// TwinCAT 3 PLC project Kid_PLC_Universal
// ProgramVersion: 3.1.4022.0
// libraries:
//   Tc2_EtherCAT, * (Beckhoff Automation GmbH)
//   Tc2_Math, * (Beckhoff Automation GmbH)
//   Tc2_MC2, * (Beckhoff Automation GmbH)
//   Tc2_System, * (Beckhoff Automation GmbH)
//   Tc2_SystemCX, * (Beckhoff Automation GmbH)
//   Tc2_Utilities, * (Beckhoff Automation GmbH)
//   Tc3_Interfaces, * (Beckhoff Automation GmbH)
//   Tc3_Module, * (Beckhoff Automation GmbH)
//   Tc2_Standard,3.3.2.0,Beckhoff Automation GmbH
// project tree:
//   DUTs/ ST_CoEdata.TcDUT, ST_CoEDataArray.TcDUT (not stored), ST_EtherCATAxis.TcDUT, ST_PointTestData.TcDUT (not stored)
//   GVLs/ GVL_DriveParameters.TcGVL (not stored), GVL_Motion.TcGVL, GVL_Hardware_IO.TcGVL, GVL_HMI.TcGVL (not stored), GVL_Index.TcGVL, GVL_IO.TcGVL (not stored), GVL_Modes.TcGVL, GVL_PLC.TcGVL (not stored), GVL_Safe_IO.TcGVL (not stored)
//   POUs/Function Blocks/ FB_CoE_ReadParamArray.TcPOU, FB_CoE_ReadParam.TcPOU (not stored), FB_CoE_WriteParamArray.TcPOU, FB_CoE_SaveParam.TcPOU, FB_EstopLED.TcPOU, FB_IntelligentFlasher.TcPOU (not stored), FB_Pulse.TcPOU, FB_SerialCom.TcPOU (not stored), FB_stCoEData_Comparison.TcPOU, FB_WriteLimits.TcPOU, FB_IgnoreLimits.TcPOU
//   POUs/Functions/ E_Custom_Trip_Codes.TcDUT (not stored), F_Scale_LR.TcPOU, F_Timed_Index_1.TcPOU (not stored), F_LimitTarget.TcPOU, F_Update_HumanReadable.TcPOU
//   POUs/ LogEvents.TcPOU (not stored), Notes.TcPOU (not stored), To_Do_List.TcPOU (not stored)
//   POUs/Programs/EtherCAT/ FB_CheckIn_EtherCAT.TcPOU, FB_EtherCATReader.TcPOU, FB_INIT_EtherCAT.TcPOU, FB_MoveAbsolute_EtherCAT.TcPOU
//   POUs/Programs/Initialize/ P1_INIT.TcPOU, P2_DriveLoad.TcPOU, P3_DriveVerification.TcPOU (not stored), P4_PowerUp.TcPOU, FB_FileCopy.TcPOU
//   POUs/Programs/Main Program/ EtherCATComs.TcPOU, MAIN.TcPOU, JoyStickMotion.TcPOU, P42_BrakeControl.TcPOU, P20_ErrorHandling.TcPOU
//   POUs/Programs/ P_AxisDataSelect.TcPOU
//   POUs/Programs/Safety Programs/ P41_SafetyHandling.TcPOU, P_Safety_Mapping.TcPOU, P_SafetyErrors.TcPOU
//   POUs/Programs/Serial/ P_EL600x.TcPOU (not stored), P_LEDstatus.TcPOU, P_Serial.TcPOU, P_SerialRemote.TcPOU (not stored)
//   POUs/Programs/Test Programs/ P_CoE_Read_Test.TcPOU (not stored), P_Drive_Save.TcPOU (not stored), P_ParameterComm.TcPOU
//   POUs/Tasks/ AxisDataTask.TcTTO (not stored), FastTask.TcTTO (not stored), PlcTask.TcTTO
// real-time tasks:
//   TASK PlcTask: cycle T#4ms, priority 20, ADS port 350
//   TASK AxisDataTask: cycle T#2ms, priority 1, ADS port 351
//   TASK FastTask: cycle T#1ms, priority 2, ADS port 352
// I/O:
//   DEVICE Device 1 (EtherCAT), AmsNetId 5.39.59.203.2.1
//     Term 1 (EK1200) [EK1200-5000 EtherCAT Power supply (2A E-Bus)]
//       Term 2 (EL6900) [EL6900, TwinSAFE PLC]
//       Term 3 (EL2904) [EL2904, 4 Ch. Safety Output 24V, 0.5A, TwinSAFE]
//         modules: Module 1 (FSOES), Module 2 (DO)
//       Term 4 (EL1008) [EL1008 8Ch. Dig. Input 24V, 3ms]
//       Term 5 (EL1904) [EL1904, 4 Ch. Safety Input 24V, TwinSAFE]
//         modules: Module 1 (FSOES)
//       Term 6 (EL2808) [EL2808 8Ch. Dig. Output 24V, 0.5A]
//       Term 7 (EL1904) [EL1904, 4 Ch. Safety Input 24V, TwinSAFE]
//         modules: Module 1 (FSOES)
//       Term 17 (EL9510) [EL9510 Power supply terminal 10V]
//       Term 18 (EL3356) [EL3356 1Ch. Ana. Input Resistor Bridge Terminal, 16bit, High Precision]
//       Term 10 (EK1110) [EK1110 EtherCAT extension]
//     Drive 11 (Unidrive M700 RFC-S) [Unidrive M700 RFC-S]
//   DEVICE Device 3 (EtherCAT Slave), AmsNetId 5.36.56.172.5.255
//   DEVICE Device 4 (EtherCAT Automation Protocol) (disabled), AmsNetId 10.4.1.1.5.1
//   DEVICE Device 6 (NOV-DP-RAM) (disabled)
// variable links:
//   TIID <-> Device 1 (EtherCAT)
//     Device 3 (EtherCAT Slave)/Outputs/AMSAddress_10/netId <-> InfoData/AmsNetId
//   Device 1 (EtherCAT) <-> Device 1 (EtherCAT)/Term 1 (EK1200)/Term 2 (EL6900)
//     Term 1 (EK1200)/Term 3 (EL2904)/Module 1 (FSOES)/RxPDO/FSOE <-> ConnectionInputs/TwinSafeGroup1.Term 3 (EL2904) - Module 1 (FSOES)_76 TxPDO
//     Term 1 (EK1200)/Term 7 (EL1904)/Module 1 (FSOES)/RxPDO/FSOE <-> ConnectionInputs/TwinSafeGroup1.Term 7 (EL1904) - Module 1 (FSOES)_78 TxPDO
//     Term 1 (EK1200)/Term 5 (EL1904)/Module 1 (FSOES)/TxPDO/FSOE <-> ConnectionOutputs/TwinSafeGroup1.Term 5 (EL1904) - Module 1 (FSOES)_77 RxPDO
//   Device 1 (EtherCAT) <-> Device 1 (EtherCAT)/Term 1 (EK1200)/Term 3 (EL2904)
//     Term 1 (EK1200)/Term 2 (EL6900)/ConnectionOutputs/TwinSafeGroup1.Term 3 (EL2904) - Module 1 (FSOES)_76 RxPDO <-> Module 1 (FSOES)/TxPDO/FSOE
//   Device 1 (EtherCAT) <-> Device 1 (EtherCAT)/Term 1 (EK1200)/Term 5 (EL1904)
//     Term 1 (EK1200)/Term 2 (EL6900)/ConnectionInputs/TwinSafeGroup1.Term 5 (EL1904) - Module 1 (FSOES)_77 TxPDO <-> Module 1 (FSOES)/RxPDO/FSOE
//   Device 1 (EtherCAT) <-> Device 1 (EtherCAT)/Term 1 (EK1200)/Term 7 (EL1904)
//     Term 1 (EK1200)/Term 2 (EL6900)/ConnectionOutputs/TwinSafeGroup1.Term 7 (EL1904) - Module 1 (FSOES)_78 RxPDO <-> Module 1 (FSOES)/TxPDO/FSOE
//   Kid_PLC_Universal/Kid_PLC_Universal Instance <-> Device 1 (EtherCAT)/Drive 11 (Unidrive M700 RFC-S)
//     FastTask Inputs/GVL_IO.kidAxis.ErrorCode <-> TxPDO5 mapping parameters/error_code
//     FastTask Inputs/GVL_IO.kidAxis.OpModeAct <-> TxPDO5 mapping parameters/modes_of_operation
//     FastTask Inputs/GVL_IO.kidAxis.P2Position <-> TxPDO5 mapping parameters/P2_Normalized
//     FastTask Inputs/GVL_IO.kidAxis.actualPos <-> TxPDO3 mapping parameters/Position actual value
//     FastTask Inputs/GVL_IO.kidAxis.pVelDem <-> TxPDO3 mapping parameters/vl_velocity_demand
//     FastTask Inputs/GVL_IO.kidAxis.statusWord <-> TxPDO3 mapping parameters/statusword
//     FastTask Inputs/GVL_IO.nAnalog_Input_Raw <-> TxPDO3 mapping parameters/#0.07.001: AnalogueInput1
//     FastTask Outputs/GVL_DriveParameters.controlWord <-> RxPDO3 mapping parameters/controlword
//     FastTask Outputs/GVL_IO.kidAxis.Denominiator1 <-> RxPDO3 mapping parameters/delta_time
//     FastTask Outputs/GVL_IO.kidAxis.Denominiator2 <-> RxPDO3 mapping parameters/delta_time_1
//     FastTask Outputs/GVL_IO.kidAxis.OpModeCMD <-> RxPDO3 mapping parameters/modes_of_operation_display
//     FastTask Outputs/GVL_IO.kidAxis.PAccel <-> RxPDO3 mapping parameters/delta_speed_Accel
//     FastTask Outputs/GVL_IO.kidAxis.pDecel <-> RxPDO3 mapping parameters/delta_speed_Decel
//     FastTask Outputs/GVL_IO.kidAxis.pVelMax <-> RxPDO3 mapping parameters/vl_target_velocity
//     PlcTask Inputs/GVL_DriveParameters.dnCurrentMagnitude <-> TxPDO5 mapping parameters/#0.04.001: CurrentMagnitude
//     PlcTask Inputs/GVL_DriveParameters.nP1_MotorThermistor <-> TxPDO3 mapping parameters/#0.03.122: P1ThermistorTemperature
//     PlcTask Inputs/GVL_IO.DriveThermalTripPercentage <-> TxPDO3 mapping parameters/#0.07.036: PercentageOfDriveThermalTripLevel
//     PlcTask Inputs/GVL_IO.bDrive_Motor_Brake_Release <-> TxPDO5 mapping parameters/#0.12.040: BcRelease
//     PlcTask Inputs/GVL_IO.stAmsAddr_Kid_1/netId <-> InfoData/AdsAddr/netId
//     PlcTask Inputs/GVL_IO.stAmsAddr_Kid_1/port <-> InfoData/AdsAddr/port
//   Kid_PLC_Universal/Kid_PLC_Universal Instance <-> Device 1 (EtherCAT)/Term 1 (EK1200)/Term 2 (EL6900)
//     FastTask Inputs/GVL_Safe_IO.bES_Local_Status <-> StandardInputs/TwinSafeGroup1.bES_Local_Status_67
//     FastTask Outputs/GVL_Safe_IO.bContactor <-> StandardOutputs/TwinSafeGroup1.bContactor_57
//     FastTask Outputs/GVL_Safe_IO.bHard_Down_Bypass_Enable <-> StandardOutputs/TwinSafeGroup1.bHard_Down_Bypass_Enable_80
//     FastTask Outputs/GVL_Safe_IO.bHard_Up_Bypass_Enable <-> StandardOutputs/TwinSafeGroup1.bHard_Up_Bypass_Enable_79
//     FastTask Outputs/GVL_Safe_IO.bPlcEstopSignal <-> StandardOutputs/TwinSafeGroup1.bPlcEstopSignal_75
//     FastTask Outputs/GVL_Safe_IO.bRelease_Load_Brake <-> StandardOutputs/TwinSafeGroup1.bRelease_Load_Brake_48
//     FastTask Outputs/GVL_Safe_IO.bRelease_Motor_Brake <-> StandardOutputs/TwinSafeGroup1.bRelease_Motor_Brake_47
//     PlcTask Inputs/GVL_IO.stAmsAddr_EL6900 <-> InfoData/AdsAddr
//     PlcTask Inputs/GVL_Safe_IO.bCom_Error <-> StandardInputs/TwinSafeGroup1.bCom_Error_54
//     PlcTask Inputs/GVL_Safe_IO.bES_Decel <-> StandardInputs/TwinSafeGroup1.bES_Decel_8
//     PlcTask Inputs/GVL_Safe_IO.bES_Error_Local <-> StandardInputs/TwinSafeGroup1.bES_Error_50
//     PlcTask Inputs/GVL_Safe_IO.bEmergency_Brake_Release_Status <-> StandardInputs/TwinSafeGroup1.bEmergency_Brake_Release_Status_73
//     PlcTask Inputs/GVL_Safe_IO.bFB_Error <-> StandardInputs/TwinSafeGroup1.bFB_Error_55
//     PlcTask Inputs/GVL_Safe_IO.bFast_Decel <-> StandardInputs/TwinSafeGroup1.bFast_Decel_25
//     PlcTask Inputs/GVL_Safe_IO.bOut_Error <-> StandardInputs/TwinSafeGroup1.bOut_Error_56
//     PlcTask Outputs/GVL_Safe_IO.bAck_Error <-> StandardOutputs/TwinSafeGroup1.bAck_Error_1
//     PlcTask Outputs/GVL_Safe_IO.bCross_Groove_Bypass_Enable <-> StandardOutputs/TwinSafeGroup1.bCross_Groove_Bypass_Enable_92
//     PlcTask Outputs/GVL_Safe_IO.bES_Restart_Local <-> StandardOutputs/TwinSafeGroup1.bES_Restart_5
//     PlcTask Outputs/GVL_Safe_IO.bEnable_Emergency_Brake_Release_Button <-> StandardOutputs/TwinSafeGroup1.bEnable_Emergency_Brake_Release_Button_59
//     PlcTask Outputs/GVL_Safe_IO.bLimit_Ultimate_Bypass_Enable <-> StandardOutputs/TwinSafeGroup1.bLimit_Ultimate_Bypass_Enable_61
//     PlcTask Outputs/GVL_Safe_IO.bMotor_Not_Moving <-> StandardOutputs/TwinSafeGroup1.bMotor_Not_Moving_60
//     PlcTask Outputs/GVL_Safe_IO.bSlack_Line_Bypass_Enable <-> StandardOutputs/TwinSafeGroup1.bSlack_Line_Bypass_Enable_91
//   Kid_PLC_Universal/Kid_PLC_Universal Instance <-> Device 1 (EtherCAT)/Term 1 (EK1200)/Term 4 (EL1008)
//     FastTask Inputs/GVL_Hardware_IO.bLoad_Brake_Feedback <-> Channel 3/Input
//     FastTask Inputs/GVL_Hardware_IO.bLocal_Deadman_State <-> Channel 7/Input
//     FastTask Inputs/GVL_Hardware_IO.bLocal_Keyswitch_Return <-> Channel 5/Input
//     PlcTask Inputs/GVL_Hardware_IO.bFan_PLC_Locked <-> Channel 1/Input
//     PlcTask Inputs/GVL_Hardware_IO.bPower_Supply_OK <-> Channel 2/Input
//     PlcTask Inputs/GVL_Hardware_IO.bUPS_BatteryReplace <-> Channel 8/Input
//   Kid_PLC_Universal/Kid_PLC_Universal Instance <-> Device 1 (EtherCAT)/Term 1 (EK1200)/Term 5 (EL1904)
//     FastTask Inputs/GVL_Safe_IO.bLimit_Ultimate <-> Module 1 (FSOES)/TxPDO/FSOE/InputChannel2
//     FastTask Inputs/GVL_Safe_IO.bSlack_Line <-> Module 1 (FSOES)/TxPDO/FSOE/InputChannel4
//     PlcTask Inputs/GVL_Safe_IO.bES1_Cir1_Local <-> Module 1 (FSOES)/TxPDO/FSOE/InputChannel1
//     PlcTask Inputs/GVL_Safe_IO.bES1_Cir2_Local <-> Module 1 (FSOES)/TxPDO/FSOE/InputChannel3
//   Kid_PLC_Universal/Kid_PLC_Universal Instance <-> Device 1 (EtherCAT)/Term 1 (EK1200)/Term 6 (EL2808)
//     PlcTask Outputs/GVL_Hardware_IO.bDeadman_Drive <-> Channel 2/Output
//     PlcTask Outputs/GVL_Hardware_IO.bES_Local_LED <-> Channel 5/Output
//     PlcTask Outputs/GVL_Hardware_IO.bEm_Brake_Release_LED <-> Channel 3/Output
//     PlcTask Outputs/GVL_Hardware_IO.bFan_Case <-> Channel 8/Output
//     PlcTask Outputs/GVL_Hardware_IO.bFan_PLC <-> Channel 7/Output
//     PlcTask Outputs/GVL_Hardware_IO.bHMI_Power <-> Channel 4/Output
//     PlcTask Outputs/GVL_Hardware_IO.bLocal_Keyswitch_Supply <-> Channel 6/Output
//     PlcTask Outputs/GVL_Hardware_IO.bMotion_LED <-> Channel 1/Output
//   Kid_PLC_Universal/Kid_PLC_Universal Instance <-> Device 1 (EtherCAT)/Term 1 (EK1200)/Term 7 (EL1904)
//     FastTask Inputs/GVL_Safe_IO.bCross_Groove <-> Module 1 (FSOES)/TxPDO/FSOE/InputChannel1
//     FastTask Inputs/GVL_Safe_IO.bLimit_Hard_Down <-> Module 1 (FSOES)/TxPDO/FSOE/InputChannel4
//     FastTask Inputs/GVL_Safe_IO.bLimit_Hard_Up <-> Module 1 (FSOES)/TxPDO/FSOE/InputChannel2
//   Kid_PLC_Universal/Kid_PLC_Universal Instance <-> Device 3 (EtherCAT Slave)
//     FastTask Inputs/GVL_IO.kidAxis.IsUltimateLimitBypassed <-> Inputs/IsUltimateLimitByPassed_5
//     FastTask Inputs/GVL_IO.kidAxis.UpdateWord_FromMom <-> Inputs/UpdateWord_FromMom_1
//     FastTask Inputs/GVL_IO.kidAxis.modeAccel_FromMom_Raw <-> Inputs/modeAccel_FromMom_Raw_4
//     FastTask Inputs/GVL_IO.kidAxis.modeDecel_FromMom_Raw <-> Inputs/ModeDecell_FromMom_Raw
//     FastTask Inputs/GVL_IO.kidAxis.modeVel_FromMom_Raw <-> Inputs/ModeVel_FromMom_Raw_3
//     FastTask Inputs/GVL_IO.kidAxis.targetpos_FromMom_Raw <-> Inputs/targetPos_FromMom_Raw_2
//     FastTask Outputs/GVL_IO.kidAxis.HomedPosition_toMom <-> Outputs/HomedPosition_toMom_2
//     FastTask Outputs/GVL_IO.kidAxis.IsHardDownLimitReached <-> Outputs/IsHardDownLimitReached_5
//     FastTask Outputs/GVL_IO.kidAxis.IsHardUpLimitReached <-> Outputs/IsHardUpLimitReached_4
//     FastTask Outputs/GVL_IO.kidAxis.IsUltimateLimitReached <-> Outputs/IsUltimateLimitReached_3
//     FastTask Outputs/GVL_IO.kidAxis.KidEstopCode <-> Outputs/EstopCode_9
//     FastTask Outputs/GVL_IO.kidAxis.Load <-> Outputs/Load_7
//     FastTask Outputs/GVL_IO.kidAxis.MotionControllerErrorCode <-> Outputs/EtherCATErrorCode_6
//     FastTask Outputs/GVL_IO.kidAxis.Speed <-> Outputs/Speed_8
//     FastTask Outputs/GVL_IO.kidAxis.UpdateWord_toMom <-> Outputs/UpdateWord_ToMom_1
//     FastTask Outputs/JoyStickMotion.JoyStickData <-> Outputs/JoyStickData

CONFIGURATION Kid_PLC_Universal
    RESOURCE PLC ON TwinCAT3
        TASK PlcTask(INTERVAL := T#4ms, PRIORITY := 20);
        PROGRAM P1_INIT WITH PlcTask : P1_INIT;
    END_RESOURCE
END_CONFIGURATION

// ---- DUTs/ST_CoEdata.TcDUT
TYPE ST_CoEdata :
STRUCT
	nIndex		: WORD;		//Index of CoE Address ex. 16#01
	nSubIndex	: BYTE;		//SubIndex of CoE Address ex. 16#01
	dwData		: DWORD;	//
	nDataLen	: UDINT;	//
END_STRUCT
END_TYPE

// ---- DUTs/ST_EtherCATAxis.TcDUT
TYPE ST_EtherCATAxis :
STRUCT
	////////EtherCAT MoeAbsolute
	AxisID : INT := 0;
	Status : FB_INIT_EtherCAT;
	//ReadStatus : FB_ReadStatus_EtherCAT := Status;
	//NcToPLC: FB_NcToPLC_Ethercat;
	axisMoveAbs : FB_MoveAbsolute_EtherCAT;
	CheckIn : FB_CheckIn_EtherCAT;
	//ParameterReader : FB_EtherCATReader;
	modeVel : DINT; //for hmi only

	// 1: System error sent from MOM
	ActiveTarget : DINT; //TARGET POSITION BEING USED INCLUDING LIMITS 
	modeTargetPos : DINT;  //target position for move
	
	modeAcc : DINT:= 2; //Maximum allowed Acceleration
	//modeJerk: UINT:= 80; //Maximum change in Accel per loop
	modeWindow : DINT:= 2000; //Allowed window for move to be complete
	leaveEnabled : BOOL := FALSE;
	isBusy : BOOL := FALSE;
	StartBit: BOOL :=FALSE;
	RawToUU: LREAL;
//Velocity mode	profile EtherCAT Actual Values


	VelDem_UU : DINT;
//Limits
	dnUpLimit : DINT;
	dnDownLimit: DINT;
	
byPassSoftUp : BOOL;
	byPassSoftDown : BOOL;
	byPassHardup : BOOL;
	byPassHardDown : BOOL;
	byPassUltimate : BOOL;
	
	UpdateWord_toMom  AT %Q* : UDINT;
	HomedPosition_toMom AT %Q* : DINT;
	IsUltimateLimitReached AT %Q* : BOOL;
	IsHardUpLimitReached AT %Q* : BOOL;
	IsHardDownLimitReached AT %Q* : BOOL;
	MotionControllerErrorCode AT %Q* :  UINT;
	 Address AT %Q*: AMSADDR;
	 Load AT %Q* : DINT;
	 Speed AT %Q* :DINT;
	 KidEstopCode AT %Q* : DINT;
	 
	 UpdateWord_FromMom AT %I* : UDINT; //UpdateWord sends boolean information every cycle for quick inputs like deadman and Estop
	 targetpos_FromMom_Raw AT %I* : DINT ; //FROM MOMt
	 modeVel_FromMom_Raw AT %I* : DINT ; //FROM MOM
	 modeAccel_FromMom_Raw AT %I* : DINT ;
	  modeDecel_FromMom_Raw AT %I* : DINT ;
	 IsUltimateLimitBypassed AT %I* : BOOL;
	
	
	
	//EtherCAT MOTION CONTROL VARIABLES
 PAccel AT %Q* : DINT  ;  //0x6048 vl_veloctity_acceleration
	 pDecel AT %Q* : DINT ; //0x6049 vl_velocity_deceleration
	 pVelMax AT %Q* : INT; // 0x6042 vl_target_velocity
	 OpModeCMD AT %Q* : USINT := 2;; // 0x6060 Page 39 MODES OF OPERATION COMMAND 2-vl velocity mode  7 = interpolated position mode
	  pVelDem	AT %I* : INT;
	 statusWord  AT %I* : BITARR16; //0x6041
	 actualPos AT %I*: DINT;// 0x6064 Position_actual_value
	 P2Position AT %I* : DINT; // Menu 3, item 129 secondary encoder position
	 actualVel AT %I*: DINT;
	 OpModeAct AT %I* : USINT; // 0x6061 Page 39 MODES OF OPERATION DISPLAY read only result of changing 0x6060
	 ErrorCode AT %I* : UINT;
	 dTime AT %Q*:  USINT := 2;
	  ResetCom : BOOL;
	SafteyReset: BOOL;
		P2Offset : DINT;
	EncoderSlop : DINT;
		Denominiator1  AT %Q* : INT:= 2;
		Denominiator2  AT %Q* : INT := 2;
		
		SlaveLock : BOOL;
END_STRUCT
END_TYPE

// ---- GVLs/GVL_Motion.TcGVL
VAR_GLOBAL
	
	

	
	bNC_Reset				:BOOL;		//Resets the NC Axis
	
	//nAxis_Status			:int;		//
	
END_VAR
VAR_GLOBAL PERSISTENT
		lrDistance_1_Motor_Rev	:LREAL := 350;		//Distance per one Motor revolution (mm)

	//NC-Encoder_P2
	//lrEncoder_P2_ScalingNum: LREAL := 0.0004;		//Scaling Factor Numerator (mm/INC)
	
	//NC-Encoder
	lrEncoder_ScalingNum	:REAL :=  0.0004;		//Scaling Factor Numerator (mm/INC)
//NC-Parameters
	rHoist_MaxVelocity		:REAL;		//Max Velocity of Motor (mm/s)
	rHoist_SelectedVelocity	:LREAL := 0;		//User selected Velocity, P36 limits to rHoist_MaxVelocity
	//rMotor_GearRatio		:REAL;		//Gearbox ratio
	
	//lrReference_Velocity	:LREAL;		//Maximum Velocity +10% (mm/s2)
	//lrMax_Acceleration		:LREAL;		//Maximum Motor Acceleration (mm/s2)
	//lrMax_Deceleration		:LREAL;		//Maximum Motor Deceleration (mm/s2)
	//lrSetup_MotorRevs_Per_Dist	:LREAL;	//Number of motor revolutions per reference distance
	//lrSetup_Ref_Distance	:LREAL;		//Reference Travel distance (mm)

	//lrDrum_Diameter			:LREAL;		//Drum diameter (mm)
	//lrWire_Diameter			:LREAL;		//Wire rope Diameter (mm)
	//lrDrum_Groove_Depth		:LREAL;		//Drum diameter groove depth (% of wire rope diameter)
	
	//lrEncoder_MTurnBits		:LREAL;		//Encoder Multiturn bits
	//lrEncoder_STurnBits		:LREAL;		//Encoder Singleturn bits
	lrDistance_1_Drum_Rev	:LREAL;		//Distance per one drum revolution (mm)
	// Delay for releasing the bDrive_Enable
	//tMotorBrake_Delay		: TIME;
END_VAR

// ---- GVLs/GVL_Hardware_IO.TcGVL
VAR_GLOBAL
	
//Locked Roter Fan Sensor
	bFan_PLC_Locked			AT %I* : BOOL;	//EL1008, IN-1, Cooling Fan Locked Rotor Sensor
	
//Load Brake Feedback
	bLoad_Brake_Feedback	AT %I*: BOOL;	//EL1008, IN-2, Check-Back from Load-Side Brake

//Keyswitch Return from Local Control
	bLocal_Keyswitch_Return	AT %I*: BOOL;	//EL1008, IN-3, Local power switch or Local Control Lockout

//Deadman_State
	bLocal_Deadman_State	AT %I*: BOOL;	//EL1008, IN-4, From Joystick DM
	
//Power Supply "OK"
	bPower_Supply_OK		AT %I*: BOOL;	//EL1008, IN-5, Tells if Local Power Supply is OK

//UPS "Ready"
	bUPS_Ready				AT %I*: BOOL;	//EL1008, IN-6, Is Local UPS unit in a "Ready" State

//UPS "Buffering"
	bUPS_Buffering			AT %I*: BOOL;	//EL1008, IN-7, Is Local UPS unit on Battery Power

//UPS "Replace Battery"
	bUPS_BatteryReplace		AT %I*: BOOL;	//EL1008, IN-8, Does the UPS Battery Need replacement

	nWeight : DINT;
	bTara : BOOL;
//OUTPUTS

	bMotion_LED				AT %Q* : BOOL;	//EL2808, OUT-1, Motion LED
	
	bDeadman_Drive			AT %Q* : BOOL;	//EL2808, OUT-2, Deadman Output to Drive Input DIO-4

	bEm_Brake_Release_LED	AT %Q* : BOOL;	//EL2808, OUT-3, Emergency Brake Release Button LED

	bHMI_Power				AT %Q* : BOOL;	//EL2808, OUT-4, HMI Power Supply

	bES_Local_LED			AT %Q*: BOOL;	//EL2808, OUT-5, Local E-Stop LED

	bLocal_Keyswitch_Supply	AT %Q*: BOOL;	//EL2808, OUT-6, Power Supply for Local Remote Pendant
	
	bFan_PLC				AT %Q*: BOOL;	//EL2808, OUT-7, PLC Cooling Fan Supply

	bFan_Case				AT %Q*: BOOL;	//EL2808, OUT-8, Case Cooling Fan Supply
	
END_VAR

// ---- GVLs/GVL_Index.TcGVL
VAR_GLOBAL
	
//Selected target with all settings

	//SelectedMoveType	: SINT;	
	
	//bMoveComplete		: BOOL;		//Move Complete		//19.050
	//rVelocity			: REAL;
	//rAccelerationTime	: REAL;
	//rDecelerationTime	: REAL;
	//rTarget				: REAL;
	//rTotalTime			: REAL;
	Home_Offset_UU : DINT;
// Save Last move commands

	nResumeMoveType		: INT;		//nMotion_Command of last executed move
	//rVelocity_Resume	: REAL;
	//rAcceleration_Resume: REAL;
	//rDeceleration_Resume: REAL;
	//rTarget_Resume 		: REAL;
	//rTimeRemaining_Resume	: REAL;
	//rAccelerationTime_Resume: REAL;
	//rDecelerationTime_Resume: REAL;
	//rRemaining_Distance	: REAL;
	
	
// Current Machinery Limits, last verified set from Axis Controller
	//dnInternal_MaxLimit	: DINT;
	//dnInternal_MinLimit	: DINT;
	
	//bResumeLastMoveEnable: BOOL;
END_VAR

VAR_GLOBAL PERSISTENT
	
	Initialized			: BOOL := FALSE;
	Admin_Max			: DINT;		//This is Maximum Admin Limit	//18.053
	Admin_Min			: DINT; 	//This is Minimum Admin Limit	//18.054
	User_Max_UU		: DINT;
	User_Min_UU		: DINT;
	//Target_Up			: DINT;		//This is a Saved UP Target		//19.051	
	//Target_Down 		: DINT;		//This is a Saved DOWN Target	//19.052
	Encoder_Offset		: DINT;		//This is saved encoder pulses for Zero Position
	Home_Offset			: DINT; 	//This is the offset for 0 value 
	Home_Switch_Offset 	: DINT;		//Offset for Axis home switch vs 0 value
	//Home_Direction		: BOOL; 	//True Means zero, False means Max
	Direction_Flipped	: BOOL ;     //This is the direction indicator, false for positive and true for reversed;
	//Admin_Max_Speed		: DINT;
	//Admin_Max_Accel		: DINT;
	Decel_For_Estop 	: DINT;
	Decel_For_DeadMan	: DINT;
END_VAR

// ---- GVLs/GVL_Modes.TcGVL
(*
//*****************************************************************Notes**********************************************************\\



  
  
//*****************************************************************Revs**********************************************************\\
   (          who            )(    Date    ) (   Rev     ) (								Disc						)
     Chris Mauban			 	2016.05.03		0.00.01		Added bDisableMotion
     Brent Miller				2016.05.26		0.00.02		Added bBrake_Test			allows user to test brakes (Motor & Load)		 								 				
	 						
	
//*****************************************************************Code**********************************************************\\
*)

VAR_GLOBAL
	
//Limit Switch Disable
	bDisable_Limit_Switch			: BOOL;	//If 'True', ignores limit switch inputs
	
//2nd Encoder Comparison test
	//bDisable_EncoderPosition_Test	: BOOL;	//If 'True', ignores encoder comparison b/w Motor & 2nd encoder
	nMotion_Command					: INT;	//Motion Command signal from HMI
	bDrive_Enable					: BOOL;	//Enable Motion from HMI
	lrDrive_Override				: LREAL; //Limit Motion Speed = 0.0 --> 100.0
	bStart_Motion					: BOOL;	//Start Loaded Motion Profile	
	
//If Drive is 'Slave'	
	//bGear_Slave_To_Master			: BOOL;	//If 'True', drive is Gearing, 'False', drive is Freerun
		
//Local Control Active
	//bLocal_Control_Active			: BOOL;	//If "True", drive is controlled by local joystick
	
//Wireless Control Active
	//bLocal_Wireless_Active			: BOOL;	//If "True", drive is controlled by Wireless Controller
	
//Local Control
	bLocal_Control					: BOOL;	//If a control is allowed Locally
	
//Remote 'MOM' Connected
	bRemote_Connected				: BOOL;	//If a remote PLC is connected

//Remote Lockout
	//bRemote_Lockout					: BOOL;	//If a remote 'Slave' or part of 3D group, and not master, don't allow independent control
	
//Brake Test
	//bBrake_Test						: BOOL;	//Enables a brake test to occur
	
//Drive Verification
	//bDrive_Verified					: BOOL;	//Has the drive been Verified
	//bDrive_Verified_Finished		: BOOL;	//Has the drive Finished Verification
//	bDrive_Save_CoE_Finished		: BOOL;	//Has the drive Finished Verification
	
//Set Home Position
//	bSetTo_0_Position				: BOOL;	//Motion Command must be set to 0
//	
//	bSafety_Enable_Forward			: BOOL;
//	bSafety_Enable_Reverse			: BOOL;
//	bDisableMotion					: BOOL;
	bDrive_Hardware_Enable			: BOOL;
//	bSetTo_Position					: BOOL;
//	rSet_Position					: REAL;
//	bSoft_Limits_Disabled			: BOOL;	//Confirmation of status of NC Soft Limits
//	bSetPositionBiasInit			: BOOL;
END_VAR	
VAR_GLOBAL PERSISTENT
	
	//Encoder is an Incremental Type
	//bEncoder_Type_Incremental		: BOOL;	//If 'True', Motor encoder is incremental

//Brake mode is Hold Control
	//bBrake_Mode_HoldControl			: BOOL;	//If 'True', opens Motor brake & holds at 0 speed
	
//Is this drive 'Master'
	bDrive_IS_Master				: BOOL;	//If 'True', drive is Master, 'False', drive is a Slave
	
//Is Secondary encoder Used?
	//bP2_Monitor_Enable				: bool;	//If 'True', runs comparison and monitors motor encoder and secondary encoder
END_VAR

// ---- POUs/Programs/Initialize/P1_INIT.TcPOU
PROGRAM P1_INIT
VAR
	nCase				: INT;
	FailCount 			: INT;
	Secondary_Encoder_ERROR : BOOL;
	maxslop : DINT;
	minslop : dint;
	//nCase_Read			: UINT;
	//nCase_Write			: UINT;
	FileOpen : FB_FileOpen;
	bNC_Parameters_Done	: BOOL;
	bCalculate_NC_Settings_Done: BOOL;
	//fbCoE_doRead		: FB_EcCoESdoRead;
	P1					: INT;
	nErrorID			: UDINT;

	fbWritePersistentData: FB_WritePersistentData;
	//RegSetValue : FB_RegSetValue;
	//VariableNames : ARRAY[1..5] OF STRING;

	
	CheckParam : STRING;
	CheckString : STRING;
	//FilePos : DINT;
	FileRead : FB_FileRead;
	//FileSeek : FB_FileSeek;
	GetLocalAMSNetID : FB_GetLocalAmsNetId;
	GetHostName : FB_GetHostName;
	ParamString : STRING(5000);
	FileClose : FB_FileClose;
	
	fbUpsPulse: FB_Pulse;
	nTestCnt: INT;
	
	NetIDString : String;
	bFileOpenErrorID : UDINT;
	bFileOpenError : BOOL;
END_VAR


GVL_IO.kidAxis.Denominiator1:=2;
GVL_IO.kidAxis.Denominiator2:=2;

bMotor_Not_Moving	:=	true;
 
nTestCnt := nTestCnt + 1;

 KidAxis.Status();//This function calls the ReadStatus of the axis.

//Run Always (Error Handling)
P20_ErrorHandling();

//Brake Control
//P42_BrakeControl(); Set in a FAST TASK

//Set bMotor_Not_Moving



//Case Statement for Sequential Initialization on Startup
CASE nCase OF

0: 
kidAxis.CheckIn.momControl := FALSE;
	FAILCOUNT := 0;
	P4_PowerUp();
	GetLocalAMSNetID(bExecute := FALSE);
	GetHostName(bExecute := FALSE);
	FileOpen(bExecute := FALSE);
	FileClose(bExecute := FALSE);
	nCase := nCase +1;
	FileRead(bExecute := FALSE);
	
1:		//Get NetID of PLC
kidAxis.P2Offset := KidAxis.actualPos - REAL_TO_DINT(KidAxis.P2Position * 8.6);
	GetLocalAMSNetID(bexecute := TRUE, AddrString => GVL_PLC.sNetID);
	IF sNetID <> '0.0.0.0.0.0' THEN 
		nCase := nCase + 1; 
		NetIDString := sNetID;
	END_IF

2: 		//Make FileName of Parameters
	GetHostName(sNetID := GVL_PLC.sNetId,
				bExecute := TRUE,
				sHostName => GVL_PLC.HostName);
	IF len(GVL_PLC.HostName) > 0 THEN
		nCase := nCase + 1;
	END_IF
3:  //get handle on parameter file
		FileOpen(sNetID :=   GVL_PLC.sNetID,//concat(Concat(Concat(Concat(concat(Concat(Concat(Concat(Concat(Concat(concat(CONCAT(BYTE_TO_STRING(stAmsAddr_Kid_1.netId[0]), '.'), BYTE_TO_STRING(stAmsAddr_Kid_1.netId[1])),'.'), BYTE_TO_STRING(stAmsAddr_Kid_1.netId[2])), '.'), BYTE_TO_STRING(stAmsAddr_Kid_1.netId[3])),  '.'), BYTE_TO_STRING(stAmsAddr_Kid_1.netId[4])), '.'), BYTE_TO_STRING(stAmsAddr_Kid_1.netId[5])),':'), WORD_TO_STRING(stAMSAddr_Kid_1.port)),
					  sPathName :=  CONCAT(CONCAT('\Hard DIsk2\ParameterFiles\', GVL_PLC.HostName), '.txt'),
					  nMode := fopen_moderead  OR FOPEN_MODETEXT,
					  ePath := PATH_GENERIC, 
					  bExecute := TRUE,
					  tTimeOut := T#3S,
					  hFile => GVL_DriveParameters.initFile,
					  bError => bFileOpenError,
					  nErrId => bFileOpenErrorID );	
					  
		IF GVL_DriveParameters.initFile <> 0 THEN
			nCase := nCase + 1;
		ELSE
				FailCount := FailCount + 1;
				IF FailCount > 1000 THEN nCase := nCase + 2; END_IF
		END_IF
//	nCase := 10000; // Jump to P30_MAIN for Virtual Programming
4:
			
			FileRead(sNetID := GVL_PLC.sNetId,
					hFile := GVL_DriveParameters.initFile,
					bExecute := TRUE,  
					pReadBuff := ADR(ParamString),
					cbReadLen := SIZEOF(ParamString),
					tTimeOut := T#3S);
			IF LEN(ParamString) > 10 AND FileRead.bBusy = FALSE THEN
			
				nErrorID := 1;
			
				CheckString := Left(ParamString, Find(ParamString, '$N')-1);
				p1 :=Find(ParamString, CheckString);
				ParamString := Right(ParamString, len(ParamString) - Len(CheckString)-1);
				CheckParam := Left(CheckString, Find(CheckString, ', '));
				CheckString := Right(CheckString, len(CheckString) - len(CheckParam) -1) ; 
				GVL_Index.Initialized := TRUE;
				IF NOT GVL_Index.Initialized THEN
					//IF Find(CheckParam, 'Home_Offset')>1 THEN GVL_Index.Home_Offset := STRING_TO_DINT(CheckString); END_IF
					//IF Find(CheckParam, 'lrEncoder_ScalingNum')>1 THEN GVL_Motion.lrEncoder_ScalingNum := STRING_TO_LREAL(CheckString); END_IF
					//IF Find(CheckParam, 'Home_Switch_Offset')>1 THEN GVL_Index.Home_Switch_Offset := STRING_TO_DINT(CheckString); END_IF
					//IF Find(CheckParam, 'Admin_Max_UU')>1 THEN GVL_Index.User_Max_UU := STRING_TO_DINT(CheckString); END_IF
					//IF Find(CheckParam, 'Admin_Min_UU')>1 THEN GVL_Index.User_Min_UU := STRING_TO_DINT(CheckString); END_IF
					//IF Find(CheckParam, 'Direction_Flipped')>1 THEN GVL_Index.Direction_Flipped := STRING_TO_BOOL(CheckString); END_IF
					//IF Find(CheckParam, 'Admin_Max')>1 AND Find(CheckParam, 'Admin_Max_UU')=0 THEN GVL_Index.Admin_Max := STRING_TO_DINT(CheckString); END_IF
					//IF Find(CheckParam, 'Admin_Min')>1 AND Find(CheckParam, 'Admin_Min_UU')=0 THEN GVL_Index.Admin_Min := STRING_TO_DINT(CheckString); END_IF
					//IF Find(CheckParam, 'lrDistance_')>1 THEN GVL_Motion.lrDistance_1_Motor_Rev := STRING_TO_DINT(CheckString); END_IF
			GVL_INDEX.Initialized := TRUE;
				//	IF GVL_Index.Home_Offset + (GVL_Index.Admin_Max_UU * LREAL_TO_INT(1/GVL_Motion.lrEncoder_ScalingNum)) <> GVL_Index.Admin_Max THEN GVL_Index.Admin_Max := GVL_Index.Home_Offset + GVL_Index.Admin_Max_UU * LREAL_TO_INT(1/GVL_Motion.lrEncoder_ScalingNum) ; END_IF
				//	IF GVL_Index.Home_Offset  + (GVL_Index.Admin_Min_UU * LREAL_TO_INT(1/GVL_Motion.lrEncoder_ScalingNum)) <> GVL_Index.Admin_Min THEN GVL_Index.Admin_Min := GVL_Index.Home_Offset  + (GVL_Index.Admin_Min_UU * LREAL_TO_INT(1/GVL_Motion.lrEncoder_ScalingNum)) ; END_IF
			END_IF
CheckString := '';
//RegSetValue(sSubKey
				CheckParam := '';
			ELSIF FileRead.bBusy = FALSE THEN
				nCase := nCase + 1;
			END_IF
				
			//END_WHILE*)
		
				//ParamString := RIGHT(ParamString, LEN(ParamString) - Len(CheckString));
			
			
		
			//IF NOT filegets.bBusy THEN filegets.bExecute := FALSE; END_IF
	
5: FileClose(sNetID := GVL_PLC.sNetId,
			 hFile := GVL_DriveParameters.initFile,
			 bExecute := TRUE);
			 nCase := 5 + (BOOL_TO_INT(NOT fileclose.bBusy) * 5);
	GVL_Index.Initialized := TRUE;
	GVL_Index.Home_Offset_UU := LREAL_TO_DINT(gvl_index.Home_Offset *GVL_Motion.lrEncoder_ScalingNum);
	kidAxis.modeWindow:= LREAL_TO_DINT(3.5/GVL_Motion.lrEncoder_ScalingNum);
	
10:	
	GVL_PLC.nDriveType := 1;
	A1_Calculate_NC_Settings();
	
	IF bCalculate_NC_Settings_Done THEN
		GVL_Safe_IO.bSafetySystem_Reset := TRUE;
		nCase := 40;
	END_IF
	
20:
	
	
	IF bNC_Parameters_Done THEN
		nCase := nCase +10;
	END_IF
	
	
		
30:
	
		nCase := nCase +10; 					//this is just for a test until parameters are verified

	P2_DriveLoad();							//Verify the drive params are correct


			nCase	:= 40;
	
	

40:
//Don't Run system until everything is setup
//	IF NOT GVL_Modes.bDrive_Verified THEN
		//						//
//	ELSE
			nCase := nCase +10;
//	END_IF



			
50:
	//Load Saved position (from powerdown store) if encoder is incremental	
	//IF GVL_Modes.bEncoder_Type_Incremental THEN
	//	P4_PowerUp.A1_Position_Restore();
	A1_Calculate_NC_Settings();				// Not needed any more because it is handled by the P36_Motion program
	//END_IF
		nCase := 10000; 
	

	
60:
//	kidAxis.Status();
//	kidAxis.Init();
//	IF KidAxis.Init.Ready THEN
//		nCase := 10000; 					//this is just for a test until parameters are verified
//	END_IF



//9999:	//Error Handling
//	GVL_PLC.udnFlyhousePLCErrorID := 16#01000 + 16#00000 + nErrorID;		//Program# + Action# + Case#
	
10000:	//Ok to Run P30_MAIN


	IF GVL_PLC.nDriveType = 1  OR GVL_PLC.nDriveType = 0 THEN
		GVL_Safe_IO.bSlack_Line_Bypass_Enable := TRUE;
		GVL_Safe_IO.bCross_Groove_Bypass_Enable := TRUE;
	END_IF
	
	//IF nTestCnt < 1000 THEN RETURN; END_IF
//	KidAxis.EncoderSlop := KidAxis.actualPos - KidAxis.P2Offset - REAL_TO_DINT(KidAxis.P2Position * 8.6);
//IF(kidAxis.EncoderSlop > MaxSlop) THEN maxslop := kidAxis.EncoderSlop; END_IF
	//IF(kidAxis.EncoderSlop < MinSlop) THEN minslop := kidAxis.EncoderSlop; END_IF

//IF ABS(kidAxis.EncoderSlop) > 10000 THEN
//	Secondary_Encoder_ERROR:=TRUE;
	//GVL_Safe_io.bContactor := FALSE;
//	ELSE
//bMotor_Not_Moving	:=	KidAxis.HomedPosition_toMom - (GVL_Index.Home_Offset -KidAxis.actualPos)/ LREAL_TO_INT(1/ GVL_Motion.lrEncoder_ScalingNum) < 2;			//Motor is not moving, PLC
fbUpsPulse(bEnable:= GVL_Hardware_IO.bUPS_Buffering, tTimeOn:= T#30MS, tTimeOff:= T#3S, bPulse=> );

fbWritePersistentData(
	NETID:= , 
	PORT:= 851, 
	START:= fbUpsPulse.bPulse OR GVL_Hardware_IO.bUPS_Buffering OR MAIN.LoopCount MOD 100000 < 500, 
	TMOUT:= T#100S, 
	MODE:= SPDM_2PASS, 
	BUSY=> , 
	ERR=> , 
	ERRID=>nErrorID );

		MAIN();	//Run P30_MAIN Program
//END_IF



END_CASE

ACTION A1_Calculate_NC_Settings:
(*
//*****************************************************************Notes**********************************************************\\
// This Action will take the user inputed parameters on the HMI and calculate the proper settings for
//	the NC controller to allow for proper motion and setup



  
  
//*****************************************************************Revs**********************************************************\\
   (          who            )(    Date    ) (   Rev     ) (								Disc						)
     Chris Mauban			 	2016.05.03		0.00.01		Added Global Error ID
	 Chris Mauban				2016.05.04		0.00.01		Removed individual cases for calculations
	 														Moved All NC_WriteParameters to A3_Write_NC_Parameters
				
     		 								 				
	 						
	
//*****************************************************************Code**********************************************************\\
*)




	bCalculate_NC_Settings_Done := TRUE;
END_ACTION

END_PROGRAM

// ---- POUs/Function Blocks/FB_Pulse.TcPOU
FUNCTION_BLOCK FB_Pulse
VAR_INPUT
	bEnable		: BOOL;		//When TRUE, bPulse will be on for tTimeOn and off for tTimeOff
	tTimeOn		: TIME;		//Time bPulse is On
	tTimeOff	: TIME;		//Time bPulse is Off
END_VAR
VAR_OUTPUT
	bPulse		: BOOL;
END_VAR
VAR
	fbTON		: TON;
	fbTOF		: TOF;
END_VAR

(*
//*****************************************************************Notes**********************************************************\\



  
  
//*****************************************************************Revs**********************************************************\\
   (          who            )(    Date    ) (   Rev     ) (								Disc						)
     Chris Mauban			 	2016.05.06		0.00.01		Initial Code
				
     		 								 				
	 						
	
//*****************************************************************Code**********************************************************\\
*)
fbTON(IN:= bEnable AND NOT fbTOF.Q, PT:= tTimeOn, Q=> , ET=> );
fbTOF(IN:= fbTON.Q, PT:= tTimeOff, Q=> , ET=> );

IF bEnable THEN
	bPulse := fbTON.M;
ELSE
	bPulse := FALSE;
END_IF

END_FUNCTION_BLOCK

// ---- POUs/Programs/Main Program/P20_ErrorHandling.TcPOU
PROGRAM P20_ErrorHandling
VAR
	GLOBAL_ERROR_STRING : STRING(200);
END_VAR


GLOBAL_ERROR_STRING := GVL_PLC.bGlobal_Error_String;

IF kidAxis.Status.Error THEN
	GVL_PLC.bGlobal_Error := TRUE;
	
END_IF

IF GVL_PLC.bGlobal_Reset THEN
	GLOBAL_ERROR_STRING := '';
	GVL_PLC.bGlobal_Error := FALSE;
	IF kidAxis.Status.STATf THEN
		GVL_Motion.bNC_Reset := TRUE;
		GVL_DriveParameters.controlWord := 128;
	END_IF

	GVL_PLC.bGlobal_Reset := FALSE;

END_IF

END_PROGRAM

// ---- POUs/Programs/Initialize/P4_PowerUp.TcPOU
PROGRAM P4_PowerUp
VAR
	
	//bSetup_Axis_Parameters_Complete	: BOOL;
	
	//fb_MC_WriteParameter: MC_WriteParameter;

	//fbCoE_WriteParamArray	:	FB_CoE_WriteParamArray;
	
	//bCoE_Enable: BOOL;
	//bCoE_WriteEnable: BOOL;
END_VAR

(*
//*****************************************************************Notes**********************************************************\\

  	The P_Drive_Verification program confirms that the drive parameters are set according to the motor that it is currently set up as.
	This will prevent any motion from occuring and throw an error if the parameters aren't set correctly.

  
  
//*****************************************************************Revs**********************************************************\\
   (          who            )(    Date    ) (   Rev     ) (								Disc						)
     Brent Miller			 	2016.04.08		0.00.01		Initial Code.
     		 								 				
	 						
	
//*****************************************************************Code**********************************************************\\
*)


//Setup the Motion Controller
//Setup User Units

//GVL_Modes.bDrive_Enable		:=	FALSE;		//Disable the Axis



//	IF bSetup_Axis_Parameters_Complete = FALSE THEN
//		P2_DriveLoad();		//	Verify that the drive parameters are correct & what drive is set up as
//	END_IF
P2_DriveLoad.A1_LoadParameters_ZipLift_CMP80M();




//System Power Control

//Set Local Keyswitch Supply power 'TRUE' unless a 'MOM' PLC is connected & taking control
IF NOT GVL_Modes.bRemote_Connected THEN
	GVL_Modes.bLocal_Control := TRUE;
ELSE
	GVL_Modes.bLocal_Control := FALSE;
END_IF


//Is local or remote control used

//IF GVL_Modes.bLocal_Control AND NOT GVL_Modes.bRemote_Connected THEN
	GVL_Hardware_IO.bLocal_Keyswitch_Supply := TRUE;
	
	//IF GVL_Hardware_IO.bLocal_Keyswitch_Return  OR GVL_HMI.bRem_SystemPowerEn AND NOT kidAxis.CheckIn.MomEstopActivated	THEN
		//GVL_Safe_IO.bContactor		:= TRUE;
		GVL_Hardware_IO.bHMI_Power	:= TRUE;
	
	//ELSElight
	
		//GVL_Safe_IO.bContactor		:= FALSE;
	//END_IF

//ELSE
//	GVL_Hardware_IO.bLocal_Keyswitch_Supply := FALSE;
//END_IF

ACTION A1_Position_Restore:

//This is for if P1 Encoder is an Incremental. 
//On the UPS powerdown, position of encoder should be saved
//On powerup position should be re-loaded into position
END_ACTION

END_PROGRAM

// ---- POUs/Programs/Initialize/P2_DriveLoad.TcPOU
PROGRAM P2_DriveLoad
VAR




	
// Loads CMP80M & M700 initial parameters.
	//CMP80M	: INT;
	//netId	: INT;
	//port	: INT;
	//bLoadParameters_Done: BOOL;
	

	
	
END_VAR



GVL_Index.Decel_For_DeadMan := 10000;
GVL_Index.Decel_For_Estop := 20000;
GVL_Motion.rHoist_MaxVelocity := 1000;
//GVL_Speeds.rAccel_With_MinLoad :=1000;
//GVL_Speeds.rDecel_With_MinLoad := 1000;
//nMotion_Command := 10;
KidAxis.modeAcc := 800;
GVL_Motion.lrDistance_1_Motor_Rev := 300;
//GVL_Motion.rMotor_GearRatio := 1;
//GVL_Motion.tMotorBrake_Delay := T#15S;
//GVL_Motion.lrDrum_Diameter := 300;
GVL_Motion.lrEncoder_ScalingNum := 0.00092327;
bLoadParameters_Done				:=	TRUE;

(*
//*****************************************************************Notes**********************************************************\\

  	The P_Drive_Verification program confirms that the drive parameters are set according to the motor that it is currently set up as.
	This will prevent any motion from occuring and throw an error if the parameters aren't set correctly.

  
  
//*****************************************************************Revs**********************************************************\\
   (          who            )(    Date    ) (   Rev     ) (								Disc						)
     Brent Miller			 	2016.04.08		0.00.01		Initial Code.
     		 								 				
	 						
	
//*****************************************************************Code**********************************************************\\


//	Has Drive already been verified?

IF NOT GVL_Modes.bDrive_Verified	THEN
		
	//This code will run if drive settings have not been verified
	//Will return a True value to bDrive_Verified
	//The HMI will need to load settings by setting a value of 1-100 in the Motor_Load_Parameters tag
	CASE GVL_HMI.Motor_Load_Parameters OF
		
	0:
		GVL_HMI.Motor_Load_Parameters	:= 1;
		A3_LoadParameters_Tracking();
		IF bLoadParameters_Done THEN
			GVL_Modes.bDrive_Verified := TRUE;
		END_IF
		
	1:
		A1_LoadParameters_ZipLift_CMP80M();
	//	GVL_HMI.Motor_Load_Parameters	:= 0;
		IF bLoadParameters_Done THEN
			GVL_Modes.bDrive_Verified := TRUE;
		END_IF
		
	2:
		A2_LoadParameters_ZipLift_FM050();	//
	//	GVL_HMI.Motor_Load_Parameters	:= 0;
		IF bLoadParameters_Done THEN
			GVL_Modes.bDrive_Verified := TRUE;
		END_IF
		
	ELSE	//if not any of the values listed above in Case statement then run this code
		//Figure out a way to trip the drive or prevent system from operating if bDrive_Verified = FALSE
		//pprasinos 6/9/2017 GVL_HMI.Drive_Status_Trip 	:=	E_Custom_Trip_Codes.System_Model_Unknown;
		
		//After the trip is Ack. then this needs to clear and set back to "OK"
		//pprasinos 6/9/2017 GVL_HMI.Drive_Status_Trip	:=	E_Custom_Trip_Codes.OK;
	
		
	END_CASE;
	
	
	
END_IF




*)

ACTION A1_LoadParameters_ZipLift_CMP80M:

GVL_Index.Decel_For_DeadMan := 10000;
GVL_Index.Decel_For_Estop := 20000;
GVL_Motion.rHoist_MaxVelocity := 1500;
//GVL_Speeds.rAccel_With_MinLoad :=1000;
//GVL_Speeds.rDecel_With_MinLoad := 1000;
//nMotion_Command := 10;
KidAxis.modeAcc := 1200;
GVL_Motion.lrDistance_1_Motor_Rev := 300;
//GVL_Motion.rMotor_GearRatio := 1;
//GVL_Motion.tMotorBrake_Delay := T#15S;
//GVL_Motion.lrDrum_Diameter := 300;
GVL_Motion.lrEncoder_ScalingNum := 0.00092327;
bLoadParameters_Done				:=	TRUE;
END_ACTION

END_PROGRAM

// ---- POUs/Programs/Main Program/MAIN.TcPOU
PROGRAM MAIN
VAR
		/////////////////////////////////////////////////////ETHERCAT
	//execute : BOOL :=FALSE;
	isdone : BOOL; 
	LoopCount : DINT;
	
	
	fbTON_Fan			: TON;
	fbCOE_Read_Safety	: FB_EcCoESdoRead;
	fbCOE_Read_DriveTemp: FB_EcCoESdoRead;
	nBuffer				: INT;
	nBufferCase			: INT;
	fbTON_FanCase		: TON;
	CaseFanDuty			: INT;
	PLCFanDuty 			:INT;
	//lrMyValue: UINT;
	checking : SINT;
	IsSlave : BOOL;
END_VAR

VAR PERSISTENT

END_VAR

//IF kidAxis.modeAccel_FromMom_Raw < 10 THEN RETURN; END_IF


checking :=1;
kidAxis.CheckIn();  //TRY Checking into MOM 
checking :=2;
JoyStickMotion();
checking :=5;
P42_BrakeControl();
checking :=3;
kidAxis.Status(); //Check drive health and Clear faults/enable drives
checking :=4;

A4_FanControl();						// Controls Hardware Fans powering on & off
checking :=6;
LogEvents();
checking :=7;
P41_SafetyHandling();
checking :=8;

kidAxis.axisMoveAbs();
checking :=9;
f_Update_HumanReadable();
checking :=10;
LoopCount := LoopCount +1;

IF GVL_HMI.MomControl_Bypass THEN
	bMotion_LED	:= LoopCount MOD 300 > 150;
END_IF

ACTION A4_FanControl:



// Turns on Case Fan if the Dynamic brake resistors get above 25%





// Turns on PLC Fan if the PLC & Safety modules get above 60 deg. C.

fbCOE_Read_Safety(
	sNetId		:= 	F_CreateAmsNetId(nIds:=GVL_IO.stAmsAddr_EL6900.netId), 
	nSlaveAddr	:= 	GVL_IO.stAmsAddr_EL6900.port,
	nSubIndex	:= 16#01, 
	nIndex		:= 16#FA80, 
	pDstBuf		:= ADR(nBuffer), 
	cbBufLen	:= SIZEOF(nBuffer), 
	bExecute	:= fbTON_Fan.Q,  );
	
MAIN.CaseFanDuty := 4 * (GVL_IO.DriveThermalTripPercentage -35); //Drive fan scales from 0 to 100% over the rane of 35-60% thermal trip percentage
		main.PLCFanDuty :=  10 *(nBuffer - 55); //plc fan scales from 0 to 100% over the rane of 55-65degC
		GVL_Hardware_IO.bFan_PLC := loopCount MOD 100 < main.PLCFanDuty  ;
GVL_Hardware_IO.bFan_Case :=  loopCount MOD 100 <MAIN.CaseFanDuty;
END_ACTION

END_PROGRAM

// ---- POUs/Programs/Main Program/JoyStickMotion.TcPOU
PROGRAM JoyStickMotion
VAR
//1/17/2013 10:28AM
	loopCount : DINT;

	DeadManOut 	: BOOL := FALSE;
	JoyStickData AT %Q*: UDINT;
;
END_VAR



	loopCount := loopCount +1;
IF GVL_IO.nAnalog_Input_Raw < GVL_IO.vMinValueCalib THEN vMinValueCalib := DINT_TO_LREAL(GVL_IO.nAnalog_Input_Raw + 1); END_IF
IF GVL_IO.nAnalog_Input_Raw > GVL_IO.vMaxValueCalib THEN vMaxValueCalib := DINT_TO_LREAL(GVL_IO.nAnalog_Input_Raw - 1); END_IF
IF loopCount MOD 1000 = 5 AND NOT GVL_Hardware_IO.bLocal_Deadman_State AND vTrim + GVL_IO.nAnalog_Input_Raw > 0 THEN vTrim := vTrim - 1; END_IF
IF loopCount MOD 1000 = 5 AND NOT GVL_Hardware_IO.bLocal_Deadman_State AND vTrim + GVL_IO.nAnalog_Input_Raw < 0 THEN vTrim := vTrim + 1; END_IF
IF GVL_IO.vTrim > 500 THEN GVL_IO.vTrim := 500; END_IF
IF GVL_IO.vTrim < -500 THEN GVL_IO.vTrim := -500; END_IF

	
IF GVL_IO.vTrim + GVL_IO.nAnalog_Input_Raw > 50 AND (DeadManOut OR KidAxis.checkIn.momControl) THEN
	GVL_IO.rJoystick_Feedback :=100 * EXPT((INT_TO_REAL(GVL_IO.nAnalog_Input_Raw + vTrim))/ vMaxValueCalib, 2);
ELSIF GVL_IO.vTrim + GVL_IO.nAnalog_Input_Raw < - 50 AND  (DeadManOut OR KidAxis.checkIn.momControl)  THEN
	GVL_IO.rJoystick_Feedback := -100 *EXPT((INT_TO_REAL(GVL_IO.nAnalog_Input_Raw + vTrim))/ vMinValueCalib, 2);
ELSIF  GVL_Hardware_IO.bLocal_Deadman_State AND ABS(vTrim + GVL_IO.nAnalog_Input_Raw)<50 THEN
	DeadManOut:= TRUE;
	GVL_IO.rJoystick_Feedback := 0;
ELSE
	DeadManOut:= FALSE;
END_IF


JoyStickData := REAL_TO_UDINT((GVL_IO.rJoystick_Feedback + 100)*100) + (32768 * BOOL_TO_DINT(GVL_Hardware_IO.bLocal_Deadman_State)) + 65536 * BOOL_TO_DINT(GVL_Hardware_IO.bLocal_Keyswitch_Return);

IF NOT GVL_HMI.MomControl_Bypass AND kidAxis.CheckIn.momControl THEN
		DeadManOut:= FALSE;
	 RETURN; 
END_IF

//Motion Allowed
GVL_Modes.bStart_Motion := TRUE;


	
	//GVL_DriveParameters.controlWord := 15;





//Use the set Velocity for the hoist

	GVL_Motion.rHoist_SelectedVelocity := GVL_Motion.rHoist_MaxVelocity;


GVL_Motion.rHoist_SelectedVelocity := GVL_Motion.rHoist_MaxVelocity * GVL_IO.rJoystick_Feedback/100;
//TESTING FOR SLOWDOWN & JOG FUNCTIONING


//Run the Jog Function Block	

IF GVL_IO.rJoystick_Feedback > 0.5 THEN
//kidAxis.modeTargetPos:=     f_LimitTarget(kidAxis.actualPos + LREAL_TO_DINT(((GVL_Motion.rHoist_SelectedVelocity  * ( ABS(GVL_Motion.rHoist_SelectedVelocity)/ kidAxis.modeAcc))))); 
	KidAxis.modeTargetPos := GVL_index.Admin_Max;
	//kidAxis.modeVel:= REAL_TO_DINT(ABS(GVL_Motion.rHoist_SelectedVelocity / 10));
ELSIF GVL_IO.rJoystick_Feedback < -0.5 THEN
	kidaxis.modeTargetPos := GVL_Index.Admin_Min;
	//kidAxis.modeVel:= REAL_TO_DINT(ABS(GVL_Motion.rHoist_SelectedVelocity / 10));
ELSE
	kidAxis.modeTargetPos:= LREAL_TO_DINT(kidAxis.actualpos);
	//kidAxis.modeVel:=0;
END_IF

END_PROGRAM

// ---- POUs/Programs/Main Program/P42_BrakeControl.TcPOU
PROGRAM P42_BrakeControl
VAR
	fbTOF_MotorBrake: TOF;
	OnHome : BOOL;
	HomeSwitchPositionON : DINT;
	enablecounter : DINT;
	HomeSwitchPositionOff : DINT;
	
	
END_VAR

(*
//*****************************************************************Notes**********************************************************\\


  
  
//*****************************************************************Revs**********************************************************\\
   (          who            )(    Date    ) (   Rev     ) (								Disc						)
     Chris Mauban			 	2016.05.05		0.00.01		Added Brake Logic for Load Brake
	 Brent Miller				2016.05.25		  0.00.02		Changed Motor Brake Logic to include a wait command before disabling motor			
     		 								 				
	 						
	
//*****************************************************************Code**********************************************************\\
*)



//Brake Logic for Motor brake	

// To DO:  	For Motor brake logic, brake should release once the drive has enabled and is energized
//			Brake should engage when Deadman button is released, wait 0.5 sec then disable the motor

		
		IF  GVL_Modes.bDrive_Enable AND kidaxis.Status.STATso AND kidaxis.status.ready THEN
				GVL_DriveParameters.controlWord := 15;
				GVL_Safe_IO.bRelease_Load_Brake := TRUE;
				IF  GVL_Hardware_IO.bLoad_Brake_Feedback THEN
					EnableCounter := ENableCounter + 1;
				END_IF
				IF EnableCounter > 20 THEN 
					GVL_Safe_IO.bRelease_Motor_Brake := TRUE;
			 		EnableCounter := 20; 
				END_IF
		ELSE
				IF EnableCounter > 0 THEN enablecounter :=0; END_IF
				GVL_Safe_IO.bRelease_Motor_Brake := FALSE;
				enablecounter := enablecounter -1;
				IF enablecounter < -50 THEN  
					enablecounter := -50; 
					IF  kidaxis.Status.STATso THEN GVL_DriveParameters.controlWord := 7; END_IF
				END_IF
		END_IF
		

IF NOT GVL_Safe_IO.bContactor  THEN GVL_Safe_IO.bRelease_Load_Brake := FALSE; GVL_Safe_IO.bRelease_Motor_Brake := FALSE; END_IF


//Brake Logic for Load Brake
//IF NOT GVL_PLC.bGlobal_Error THEN
//	GVL_Safe_IO.bRelease_Load_Brake := TRUE;
//ELSE
//	GVL_Safe_IO.bRelease_Load_Brake := FALSE;
//END_IF

IF GVL_Safe_IO.bCross_Groove AND NOT OnHome THEN
	HomeSwitchPositionON := KidAxis.actualPos;
	OnHome := TRUE;
ELSIF NOT GVL_SAFE_IO.bCross_Groove AND ONHOME THEN
	HomeSwitchPositionOFF := KidAxis.actualPos;
	OnHome := FALSE;
END_IF
kidAxis.CheckIn.Home_Tripped := OnHome;

ACTION A1_BrakeTest:
(*
	This program will allow the technician to test the functionality of each of the brakes.
	When in "Test" mode, both brakes will engage (not-energized) regardless of system status
	- operator will then be allowed to manually release one brake at a time (momentary release). This allows the operator to check functionality & load holding ability
	- 

*)
END_ACTION

END_PROGRAM

// ---- POUs/Programs/Safety Programs/P41_SafetyHandling.TcPOU
PROGRAM P41_SafetyHandling
VAR
	ByPassCounter : DINT;
//	fbIntelligentFlasher: FB_IntelligentFlasher;
	//bFlasher: BOOL;
	//bFlasher_Enable: BOOL;
	nCase: INT;
	fbTON: TON;
	nErrorID: INT;
	//fb_ES_LED: FB_Pulse;
	bTS_Reset: BOOL;
	fbClosetLED: FB_EstopLED;
END_VAR

IF(GVL_Safe_IO.bHard_Down_Bypass_Enable OR GVL_Safe_IO.bHard_Up_Bypass_Enable OR 
	GVL_Safe_IO.bLimit_Ultimate_Bypass_Enable OR GVL_HMI.MomControl_Bypass OR bLimit_Software_Bypass) THEN
	ByPassCounter := ByPassCounter + 1;
		IF(ByPassCOunter > 200000) or not GVL_Hardware_IO.bLocal_Keyswitch_Return THEN 
			bLimit_Software_Bypass := FALSE;
			GVL_Safe_IO.bHard_Down_Bypass_Enable := FALSE;
 			GVL_Safe_IO.bHard_Up_Bypass_Enable := FALSE;
			GVL_Safe_IO.bLimit_Ultimate_Bypass_Enable := FALSE;
  			GVL_HMI.MomControl_Bypass := FALSE;
			ByPassCounter := 200000;
		END_IF
	ELSE
		ByPassCounter :=0;
END_IF


GVL_Hardware_IO.bLocal_Keyswitch_Supply := TRUE;		//if not locked out or remote connected, then turn on keyswitch supply
			IF (GVL_Hardware_IO.bLocal_Keyswitch_Return OR GVL_io.kidAxis.CheckIn.momControl) AND 
			   ( NOT kidAxis.CheckIn.MomEstopActivated OR kidAxis.CheckIn.ResetSaftey) AND 
				(GVL_SAfe_IO.bLimit_Ultimate OR GVL_Safe_IO.bLimit_Ultimate_Bypass_Enable)	THEN
					GVL_Safe_IO.bContactor := TRUE;						//turn on contactor
					GVL_HardWare_IO.bHMI_Power := TRUE;		//turn on HMI Screen
			//		GVL_Modes.bDrive_Enable := TRUE;			
			ELSE
				GVL_Safe_IO.bContactor := FALSE;		//turn off contactor
			
				GVL_Modes.bDrive_Enable := FALSE;
			END_IF
			
	IF kidAxis.Status.STATf THEN GVL_Safe_IO.bContactor := False; END_IF
	
	GVL_Safe_IO.bPlcEstopSignal := GVL_Safe_IO.bES1_Cir1_Local AND GVL_Safe_IO.bES1_Cir2_Local;
//EStop LED
	A1_EStop_LED();

//Safety System Reset sequence
	A2_SafetyReset();
	
//P2 Encoder Comparison
	A4_P2Comparison();	

//Turn on Emergency Brake Release LED when Button is Enabled
	IF GVL_Hardware_IO.bUPS_Buffering THEN
		bEnable_Emergency_Brake_Release_Button := TRUE;
		GVL_HardWare_IO.bHMI_Power := FALSE;	
		bEm_Brake_Release_LED := 1;
		
	ELSE 
		bEnable_Emergency_Brake_Release_Button := FALSE;
		bEm_Brake_Release_LED := 0;
	END_IF


	
P_Safety_Mapping();
P_SafetyErrors();
(*
GVL_Modes.bSafety_Enable_Forward 	:= (GVL_Safe_IO.bLimit_Hard_Up OR GVL_Safe_IO.bHard_Up_Bypass_Enable)
										AND (GVL_Safe_IO.bCross_Groove OR GVL_Safe_IO.bCross_Groove_Bypass_Enable); //Belt Driven = Prox
										
	GVL_Modes.bSafety_Enable_Reverse	:= (GVL_Safe_IO.bLimit_Hard_Down OR GVL_Safe_IO.bHard_Down_Bypass_Enable)
										AND (GVL_Safe_IO.bSlack_Line OR GVL_Safe_IO.bSlack_Line_Bypass_Enable);		//Belt Driven = Prox
*)

ACTION A1_EStop_LED:
(*
//*****************************************************************Notes**********************************************************\\



  
  
//*****************************************************************Revs**********************************************************\\
   (          who            )(    Date    ) (   Rev     ) (								Disc						)
     Chris Mauban			 	2016.05.06		0.00.01		Initial Code
				
     		 								 				
	 						
	
//*****************************************************************Code**********************************************************\\
*)
fbClosetLED(bEstopSignal:= GVL_Safe_IO.bES1_Cir1_Local AND GVL_Safe_IO.bES1_Cir2_Local, bSafetySystemSignal:= GVL_Safe_IO.bES_Decel, bLEDOutput=> GVL_Hardware_IO.bES_Local_LED);
END_ACTION

ACTION A2_SafetyReset:
(*
//*****************************************************************Notes**********************************************************\\



  
  
//*****************************************************************Revs**********************************************************\\
   (          who            )(    Date    ) (   Rev     ) (								Disc						)
     Chris Mauban			 	2016.05.05		0.00.01		Removed HardUp/Dn Restarts, removed If Statements.  Using an Else
	 														will always force a No Reset
															Added Case Statement so the rising edge of the Reset will Reset Safety System Errors
															and reset Safe Estop FB.
				
     		 								 				
	 						
	
//*****************************************************************Code**********************************************************\\
*)




//SAFETY OUTPUTS

//Ouput to safety program
IF bSafetySystem_Reset THEN
	bTS_Reset := TRUE;
GVL_Safe_IO.bAck_Error	:=	TRUE;
END_IF

CASE nCase OF
	0: //Wait for Rising Edge of Reset
		IF bTS_Reset THEN
			fbTON(IN:= FALSE, PT:= T#500MS, Q=> , ET=> );
			nErrorID := 0;
			nCase := nCase + 10;
		END_IF

		
	10: //Reset System Errors
		fbTON(IN:= TRUE, PT:= T#500MS, Q=> , ET=> ); //Allow 500ms to Reset System Errors
		GVL_PLC.bSafetyErrAckInput 	:=	TRUE;
		IF NOT GVL_PLC.bSafetyError THEN
			GVL_PLC.bSafetyErrAckInput	:=	FALSE;
			fbTON(IN:= FALSE, PT:= T#500MS, Q=> , ET=> );			
			nCase := nCase + 10;
		END_IF
		IF fbTON.Q THEN	//Unable to Reset Safety System
			nErrorID := nCase;
			nCase := 9999;
		END_IF
	
	20: //Reset All Estop Function Block
		fbTON(IN:= TRUE, PT:= T#2000MS, Q=> , ET=> ); //Allow 500ms to Reset Estop Function Block
		GVL_PLC.bLocalEstopRestart	:= TRUE;
		nCase := nCase + 10;
		
	30: 
		fbTON(IN:= TRUE ); //Allow 500ms to Reset Estop Function Block
		GVL_PLC.bLocalEstopRestart	:= FALSE;
		nCase := nCase + 10;
		GVL_Safe_IO.bAck_Error	:=	FALSE;
		
	40:
		fbTON(IN:= TRUE ); //Allow 500ms to Reset Estop Function Block
		IF GVL_Safe_IO.bES_Local_Status THEN	
			fbTON(IN:= FALSE, PT:= T#2000MS, Q=> , ET=> );
			nCase := nCase + 10;
		ELSE
			IF fbTON.Q THEN	//Unable to Reset Estop Function Block
				nErrorID := nCase;
				nCase := 9999;
			ELSE
				nCase := nCase - 20; //Toggle Reset Again
			END_IF
		END_IF
		
	50: //Reset All Estop Function Block
		fbTON(IN:= TRUE, PT:= T#2000MS, Q=> , ET=> ); //Allow 500ms to Reset Estop Function Block

		nCase := nCase + 10;
		
	60: 
		fbTON(IN:= TRUE ); //Allow 500ms to Reset Estop Function Block

		nCase := nCase + 10;
		
	70: //Reset External Estop Function Block
		fbTON(IN:= TRUE ); //Allow 500ms to Reset Estop Function Block
		
			IF fbTON.Q THEN	//Unable to Reset Estop Function Block
				nErrorID := nCase;
				nCase := 9999;
			ELSE
				nCase := nCase - 20; //Toggle Reset Again
			END_IF
	
		
	9999: //Error Handling
		//GVL_PLC.udnFlyhousePLCErrorID := DINT_TO_UDINT(16#41000 + 16#100 + nCase);	//Program# + Action# + Case#
		nCase := 10000;
		
	10000:
		GVL_PLC.bSafetyErrAckInput 		:= FALSE;
		GVL_PLC.bLocalEstopRestart		:= FALSE;
		bTS_Reset						:= FALSE;
		IF NOT bSafetySystem_Reset THEN
			nCase := 0;
			ELSE
			 bSafetySystem_Reset := FALSE;
		END_IF
END_CASE
END_ACTION

ACTION A3_SafetyStatus:
(*
//*****************************************************************Notes**********************************************************\\



  
  
//*****************************************************************Revs**********************************************************\\
   (          who            )(    Date    ) (   Rev     ) (								Disc						)
     Chris Mauban			 	2016.05.06		0.00.01		Initial Code
	 Brent Miller				2016.06.15		0.00.02		Added nSafetySystem_Status to safety system readouts so 1 var. could be
															used to tell the status of all of the safety system components. Currently
															does not operate properly.			
     		 								 				
	 						
	
//*****************************************************************Code**********************************************************\\
*)
//TO-DO: (BAM) The nSafetySystem_Status does not update with the correct value

//Estop Function Block
IF NOT GVL_Safe_IO.bES_Local_Status THEN
	GVL_Safe_IO.nSafetySystem_Status := 0;//System OK
	IF NOT GVL_Safe_IO.bES1_Cir1_Local OR NOT GVL_Safe_IO.bES1_Cir2_Local THEN
		GVL_Safe_IO.nSafetySystem_Status := 1;//Local Estop Pressed
	ELSIF NOT bLimit_Ultimate THEN
		GVL_Safe_IO.nSafetySystem_Status := 2;//Ultimate LIMIT Triggered
	ELSIF NOT bPlcEstopSignal THEN
		GVL_Safe_IO.nSafetySystem_Status := 3;//Plc Estop
	ELSE //Motor did not stop after 500ms when the following triggered
		IF GVL_Safe_IO.bSlack_Line THEN
			GVL_Safe_IO.nSafetySystem_Status := 4;//Slack Line
		ELSIF GVL_Safe_IO.bLimit_Hard_Down THEN
			GVL_Safe_IO.nSafetySystem_Status := 5;//Hard Down Limit
		ELSIF GVL_Safe_IO.bLimit_Hard_Up THEN
			GVL_Safe_IO.nSafetySystem_Status := 6;//Hard Up Limit
		ELSIF GVL_Safe_IO.bCross_Groove THEN
			GVL_Safe_IO.nSafetySystem_Status := 7;//Gross Groove
		END_IF
	END_IF
END_IF

//Safety System Comm Check
IF GVL_Safe_IO.bCom_Error THEN
	GVL_Safe_IO.nSafetySystem_Status := 20;//Safety System Comm Error
ELSIF GVL_Safe_IO.bAck_Error THEN
	GVL_Safe_IO.nSafetySystem_Status := 21;//Safety System Acknolegment Error
ELSIF GVL_Safe_IO.bES_Error_Local THEN
	GVL_Safe_IO.nSafetySystem_Status := 22;//Local E-Stop FB Error
ELSE
	GVL_Safe_IO.nSafetySystem_Status := 0;//System OK
END_IF
//Continue this for all of the function blocks in the safety system

//Contactor


//Load Brake

//Motor Brake
END_ACTION

ACTION A4_P2Comparison:

//PPRASINOS 6/5/2017//IF GVL_Modes.bP2_Monitor_Enable THEN
//PPRASINOS 6/5/2017//	IF kidAxis.NcToPlc.ActPos > (kidAxis_P2.NcToPlc.ActPos + GVL_Safe_IO.nP2_EncoderWindow) THEN

	//Run routine, issue fast stop, then set Motion Command to 0, issue error, and remove "PLC_Estop"
	//possibly add a time delay for triggering the error
	
//PPRASINOS 6/5/2017//	ELSIF kidAxis.NcToPlc.ActPos < (kidAxis_P2.NcToPlc.ActPos - GVL_Safe_IO.nP2_EncoderWindow) THEN
	
	//Run routine, issue fast stop, then set Motion Command to 0, issue error, and remove "PLC_Estop"
	
	
//PPRASINOS 6/5/2017//	END_IF

	
//PPRASINOS 6/5/2017//END_IF
END_ACTION

END_PROGRAM

// ---- POUs/Function Blocks/FB_EstopLED.TcPOU
FUNCTION_BLOCK FB_EstopLED
VAR_INPUT
	bEstopSignal : BOOL;
	bSafetySystemSignal : BOOL;
END_VAR
VAR_OUTPUT
	bLEDOutput : BOOL;
END_VAR
VAR
	tOnBlinkTime : TIME;
	nNumOfOnBlinks : INT;
	tLEDOffTime : TIME;
	fbLEDPulse: FB_Pulse;
	fbBlinkPulse: FB_Pulse;
	bBlinkEn: BOOL;
	tTotalTimeOn: TIME;
	tOffBlinkTime: TIME;
END_VAR

IF NOT bEstopSignal THEN
	tOnBlinkTime := T#250MS;
	tOffBlinkTime := T#250MS;
	nNumOfOnBlinks := 3;
	tLEDOffTime := T#1000MS;
	bBlinkEn := TRUE;
	bLEDOutput := fbBlinkPulse.bPulse;	
ELSIF NOT bSafetySystemSignal THEN
	tOnBlinkTime := T#1000MS;
	tOffBlinkTime := T#250MS;
	nNumOfOnBlinks := 1;
	tLEDOffTime := T#1000MS;
	bBlinkEn := TRUE;
	bLEDOutput := fbBlinkPulse.bPulse;	
ELSE
	bLEDOutput := TRUE;	
	bBlinkEn := FALSE;
END_IF

tTotalTimeOn := DINT_TO_TIME((TIME_TO_DINT(tOnBlinkTime) * (nNumOfOnBlinks)) + (TIME_TO_DINT(tOffBlinkTime) * (nNumOfOnBlinks - 1)));
fbLEDPulse(bEnable:= bBlinkEn, tTimeOn:= tTotalTimeOn, tTimeOff:= tLEDOffTime, bPulse=> );
fbBlinkPulse(bEnable:= fbLEDPulse.bPulse, tTimeOn:= tOnBlinkTime, tTimeOff:= tOffBlinkTime, bPulse=> );

END_FUNCTION_BLOCK

// ---- POUs/Programs/Safety Programs/P_Safety_Mapping.TcPOU
PROGRAM P_Safety_Mapping
VAR
	fbF_Trig: F_TRIG;
END_VAR






//	GVL_PLC.bSafetySystemResetRequired := TRUE;


//IF GVL_Safe_IO.bAck_Error THEN
//	GVL_PLC.bSafetySystemResetRequired := FALSE;
//END_IF

//Comms to TwinSAFE
GVL_Safe_IO.bES_Restart_Local 		:= GVL_PLC.bLocalEstopRestart ;
GVL_Safe_IO.bAck_Error				:= GVL_PLC.bSafetyErrAckInput ;
//GVL_Safe_IO.bExternalEstopEn 		:= GVL_PLC.bExternalEstopEnInput;
//GVL_Safe_IO.bES_Restart_External	:= GVL_PLC.bExternalEstopRestart;


//Comms to Ethercat Slave Network

END_PROGRAM

// ---- POUs/Programs/Safety Programs/P_SafetyErrors.TcPOU
PROGRAM P_SafetyErrors
VAR
END_VAR

IF GVL_Safe_IO.bCom_Error OR 
		GVL_Safe_IO.bFB_Error OR
		GVL_Safe_IO.bOut_Error  THEN
	GVL_PLC.bSafetyError := TRUE;
END_IF





IF GVL_Safe_IO.bAck_Error THEN
	GVL_PLC.bSafetyError := FALSE;
END_IF

END_PROGRAM

// ---- POUs/Functions/F_Update_HumanReadable.TcPOU
FUNCTION F_Update_HumanReadable : BOOL
VAR_INPUT
END_VAR
VAR
	CheckVar : DINT;
	GVL_KidAxis: INT;
END_VAR

IF GVL_Motion.lrEncoder_ScalingNum = 0 THEN RETURN; END_IF
IF GVL_INDEX.Direction_Flipped THEN
	GVL_DriveParameters.Normalized_Position := (GVL_Index.Home_Offset -KidAxis.actualPos)/ LREAL_TO_INT(1/ GVL_Motion.lrEncoder_ScalingNum);
ELSE
	GVL_DriveParameters.Normalized_Position := (KidAxis.actualPos - GVL_Index.Home_Offset)/ LREAL_TO_INT(1/ GVL_Motion.lrEncoder_ScalingNum);
END_IF


GVL_DriveParameters.Normalized_Acceleration := (KidAxis.modeAcc * LREAL_TO_INT(GVL_Motion.lrDistance_1_Motor_Rev))/120;
//GVL_DriveParameters.Normalized_Min_Limit := GVL_Index.Admin_Min / LREAL_TO_INT(1/ GVL_Motion.lrEncoder_ScalingNum);
//GVL_DriveParameters.Normalized_Max_Limit := GVL_Index.Admin_Max / LREAL_TO_INT(1/GVL_Motion.lrEncoder_ScalingNum);

KidAxis.HomedPosition_toMom := GVL_DriveParameters.Normalized_Position;

CheckVar := GVL_DriveParameters.targetpos_FromMom;

CheckVar := F_LimitTarget((GVL_DriveParameters.targetpos_FromMom * 3020) + GVL_Index.Home_Offset);


///GVL_DriveParameters.modeVel_FromMom := 1 + (LREAL_TO_INT(KidAxis.modeVel_FromMom_Raw * 1000) / LREAL_TO_INT(1/ GVL_Motion.lrEncoder_ScalingNum));
///GVL_DriveParameters.modeAccel_FromMom := 1 + (LREAL_TO_INT(KidAxis.modeAccel_FromMom_Raw * 1000) /LREAL_TO_INT(1/ GVL_Motion.lrEncoder_ScalingNum));
///GVL_DriveParameters.modeDecel_FromMom := 1 + (LREAL_TO_INT(KidAxis.modeDecel_FromMom_Raw * 1000) /LREAL_TO_INT(1/ GVL_Motion.lrEncoder_ScalingNum));
GVL_DriveParameters.modeVel_FromMom := KidAxis.modeVel_FromMom_Raw;
GVL_DriveParameters.modeAccel_FromMom := 1 + KidAxis.modeAccel_FromMom_Raw;
GVL_DriveParameters.modeDecel_FromMom := 1 + KidAxis.modeDecel_FromMom_Raw;
GVL_DriveParameters.targetpos_FromMom := KidAxis.targetpos_FromMom_Raw;
KidAxis.velDem_UU := LREAL_TO_DINT(KidAxis.pVelDem * GVL_Motion.lrDistance_1_Motor_Rev);

	GVL_HMI.GlobalEstopCode := BOOL_TO_UDINT(kidAxis.CheckIn.SafteyTripped) * ULINT_TO_UDINT(+ (BOOL_TO_ULINT(kidAxis.CheckIn.safteyTripped) * (BOOL_TO_ULINT(kidAxis.CheckIn.momControl) * 1 +
					BOOL_TO_ULINT(kidAxis.CheckIn.Rmt_DeadManPressed) * 2 +
					BOOL_TO_ULINT(NOT kidAxis.Status.voltageEnabled) * 4 + 
					BOOL_TO_ULINT(kidAxis.Status.switchOnDisabled) * 8 + 
					BOOL_TO_ULINT(NOT bPlcEstopSignal) * 16 + 
					BOOL_TO_ULINT(NOT GVL_Safe_IO.bLimit_Ultimate) * 32 + 
					BOOL_TO_ULINT(NOT GVL_Safe_IO.bMotor_Not_Moving) * 64 + 
					BOOL_TO_ULINT(GVL_Safe_IO.bContactor) * 128 + 
					BOOL_TO_ULINT(NOT GVL_Safe_IO.bRelease_Load_Brake) * 256 + 
					BOOL_TO_ULINT(NOT GVL_Safe_IO.bRelease_Motor_Brake) * 512 + 
					BOOL_TO_ULINT(GVL_Safe_IO.bSafetySystem_Reset) * 1024 )));
					
					//IF GVL_IO.kidAxis.HomeOffset_UU_W <>0 AND GVL_IO.kidAxis.HomeOffset_UU_W <> GVL_Index.Home_Offset / LREAL_TO_INT(1/GVL_Motion.lrEncoder_ScalingNum) THEN
					//	GVL_Index.Home_Offset_UU := GVL_IO.kidAxis.HomeOffset_UU_W;
						//GVL_Index.Home_Switch_Offset := GVL_Index.Home_Switch_Offset + (GVL_Index.Home_Offset_UU * LREAL_TO_INT((1/GVL_Motion.lrEncoder_ScalingNum)) -GVL_Index.Home_Offset); 
					//	IF GVL_Index.Home_Offset_UU <> 0 THEN GVL_Index.Home_Offset := GVL_IO.kidAxis.HomeOffset_UU_W * LREAL_TO_INT(1/GVL_Motion.lrEncoder_ScalingNum); END_IF
					//END_IF
	GVL_IO.kidAxis.KidEstopCode := GVL_HMI.GlobalEstopCode;
	GVL_IO.KidAxis.MotionControllerErrorCode := GVL_IO.kidAxis.ErrorCode;
	//GVL_IO.kidAxis.HomeOffset_UU_R := GVL_Index.Home_Offset_UU;
	GVL_IO.kidAxis.Speed := kidaxis.pVelDem;
	GVL_IO.kidAxis.Load := DINT_TO_INT(GVL_DriveParameters.dnCurrentMagnitude);
	GVL_IO.kidAxis.IsUltimateLimitReached := NOT GVL_Safe_IO.bLimit_Ultimate;
	
	GVL_IO.kidAxis.IsHardUpLimitReached := NOT GVL_Safe_IO.bLimit_Hard_Up ;
	GVL_IO.kidAxis.IsHardDownLimitReached := NOT GVL_Safe_IO.bLimit_Hard_Down ;

	
	
	
	
	IF GVL_HMI.Set_User_Home THEN
		GVL_Index.Home_Offset := KidAxis.actualPos;
		GVL_HMI.Set_User_Home := FALSE;
	END_IF
//	IF GVL_io.kidAxis.CheckIn.SetSoftDown THEN
//		IF GVL_INDEX.direction_Flipped THEN GVL_Index.Admin_Max := GVL_IO.kidAxis.actualPos; ELSE GVL_Index.Admin_Min := GVL_IO.kidAxis.actualPos; END_IF
//	END_IF
	
//	IF GVL_io.kidAxis.CheckIn.SetSoftUp THEN
//		IF GVL_INDEX.direction_Flipped THEN GVL_Index.Admin_Min := GVL_IO.kidAxis.actualPos; ELSE GVL_Index.Admin_Max := GVL_IO.kidAxis.actualPos; END_IF
//	END_IF

END_FUNCTION

// ---- POUs/Functions/F_LimitTarget.TcPOU
FUNCTION F_LimitTarget : DINT //used to translate EtherCAT communication from RAW variables to Kid Variables

VAR_INPUT
	Target : DINT;
END_VAR
VAR
	CorrectedTarget : DINT;
	ho: INT;
	Resulting_Max : DINT;
	Resulting_Min : DINT;
	posi: INT;
END_VAR


CorrectedTarget := GVL_index.Home_Offset;
CorrectedTarget := KidAxis.actualPos;
CorrectedTarget := KidAxis.HomedPosition_toMom;
CorrectedTarget := Target ;

IF KidAxis.IsUltimateLimitBypassed THEN 
	F_LimitTarget := Target;
	RETURN;
END_IF

IF SetAdminMax THEN GVL_Index.Admin_Max := KidAxis.actualPos; SetAdminMax := FALSE; END_IF
IF SetAdminMin THEN GVL_Index.Admin_Min := KidAxis.actualPos; SetAdminMin := FALSE;END_IF	
IF SetUserMax AND KidAxis.HomedPosition_toMom > GVL_Index.User_Max_UU THEN GVL_Index.User_Max_UU := KidAxis.HomedPosition_toMom; SetUserMax:=FALSE; END_IF
IF SetUserMin AND KidAxis.HomedPosition_toMom > GVL_Index.User_Min_UU THEN GVL_Index.User_Min_UU := KidAxis.HomedPosition_toMom; SetUserMin:= FALSE; END_IF

IF GVL_HMI.BlowOutLimits THEN
	GVL_Index.Admin_Max := 2147483647;
	GVL_Index.Admin_Min := -2147483648;
	GVL_Index.User_Max_UU := 32000;
	GVL_Index.User_Min_UU := -32000;
	GVL_HMI.BlowOutLimits := FALSE;
END_IF

		
//ADMIN LIMITS
 
IF NOT GVL_Index.Direction_Flipped THEN
	IF GVL_Index.Home_Offset + (GVL_Index.User_Min_UU *LREAL_TO_INT(1/ GVL_Motion.lrEncoder_ScalingNum))< GVL_Index.admin_Min THEN GVL_Index.User_Min_UU := (GVL_Index.Admin_Min -GVL_Index.Home_Offset)/LREAL_TO_INT(1/ GVL_Motion.lrEncoder_ScalingNum); END_IF
	IF GVL_Index.Home_Offset + (GVL_Index.User_Max_UU *LREAL_TO_INT(1/ GVL_Motion.lrEncoder_ScalingNum))> GVL_Index.admin_Max THEN GVL_Index.User_Max_UU := (GVL_Index.Admin_Max -GVL_Index.Home_Offset)/LREAL_TO_INT(1/ GVL_Motion.lrEncoder_ScalingNum); END_IF
	Resulting_Max := GVL_Index.Home_Offset + (GVL_Index.User_Max_UU *LREAL_TO_INT(1/ GVL_Motion.lrEncoder_ScalingNum));
	Resulting_Min := GVL_Index.Home_Offset + (GVL_Index.User_Min_UU *LREAL_TO_INT(1/ GVL_Motion.lrEncoder_ScalingNum));
	IF CorrectedTarget > KidAxis.actualPos AND  (NOT GVL_Safe_IO.bLimit_Hard_Up AND NOT GVL_Safe_IO.bHard_Up_Bypass_Enable) THEN CorrectedTarget := KidAxis.actualPos; END_IF
	IF CorrectedTarget < KidAxis.actualPos AND  (NOT GVL_Safe_IO.bLimit_Hard_down AND NOT GVL_Safe_IO.bHard_DOWN_Bypass_Enable) THEN CorrectedTarget := KidAxis.actualPos; END_IF
ELSE
	IF GVL_Index.Home_Offset + (GVL_Index.User_Max_UU *LREAL_TO_INT(1/ GVL_Motion.lrEncoder_ScalingNum))< GVL_Index.admin_Min THEN GVL_Index.User_Max_UU := (GVL_Index.Admin_Min -GVL_Index.Home_Offset)/LREAL_TO_INT(1/ GVL_Motion.lrEncoder_ScalingNum); END_IF
	IF GVL_Index.Home_Offset + (GVL_Index.User_Min_UU *LREAL_TO_INT(1/ GVL_Motion.lrEncoder_ScalingNum))> GVL_Index.admin_Max THEN GVL_Index.User_Min_UU := (GVL_Index.Admin_Max -GVL_Index.Home_Offset)/LREAL_TO_INT(1/ GVL_Motion.lrEncoder_ScalingNum); END_IF
	Resulting_Min:= GVL_Index.Home_Offset + (GVL_Index.User_Max_UU *LREAL_TO_INT(1/ GVL_Motion.lrEncoder_ScalingNum));
	Resulting_Max := GVL_Index.Home_Offset + (GVL_Index.User_Min_UU *LREAL_TO_INT(1/ GVL_Motion.lrEncoder_ScalingNum));
	IF CorrectedTarget < KidAxis.actualPos AND  (NOT GVL_Safe_IO.bLimit_Hard_Up AND NOT GVL_Safe_IO.bHard_Up_Bypass_Enable) THEN CorrectedTarget := KidAxis.actualPos; END_IF
	IF CorrectedTarget > KidAxis.actualPos AND  (NOT GVL_Safe_IO.bLimit_Hard_down AND NOT GVL_Safe_IO.bHard_DOWN_Bypass_Enable) THEN CorrectedTarget := KidAxis.actualPos; END_IF
END_IF

IF NOT bLimit_Software_Bypass THEN
	IF CorrectedTarget > Resulting_Max THEN CorrectedTarget := Resulting_Max; END_IF
	IF CorrectedTarget < Resulting_Min THEN CorrectedTarget := Resulting_Min ; END_IF
END_IF

kidAxis.ActiveTarget := CorrectedTarget;
F_LimitTarget := CorrectedTarget;

RETURN ;

END_FUNCTION

// ---- POUs/Function Blocks/FB_CoE_ReadParamArray.TcPOU
FUNCTION_BLOCK FB_CoE_ReadParamArray
VAR_INPUT
	bExecute: BOOL;
	sNetId: T_AmsNetID;
	nSlaveAddr: UINT;
	tTimeout: TIME;
	nSizeOfArr: USINT;
END_VAR
VAR_OUTPUT
	bBusy: BOOL;
	bDone: BOOL;
	/// Current ST_CoEDataArray Array Location being Read
	nCurArrLoc: INT;
	bError: BOOL;
	/// http://infosys.beckhoff.com/content/1033/tcadscommon/html/ads_returncodes.htm
	nErrorID: UDINT;
END_VAR
VAR
	fbCoE_Read: FB_EcCoESdoRead;
	nCase: INT;
	nIndex: INT;
END_VAR
VAR_IN_OUT
	stCoEDataArray: ST_CoEDataArray;
END_VAR

(*++++++++++++++ CoE communication ++++++++++++++++++++++*)
fbCoE_Read.sNetId		:= sNetId;
fbCoE_Read.nSlaveAddr 	:= nSlaveAddr;
fbCoE_Read.tTimeout		:= tTimeout;

//Automatically Resets FB if bExecute is False
IF NOT bExecute THEN
	nCase 		:= 0;
	bError 		:= FALSE;
	bBusy 		:= FALSE;
	bDone 		:= FALSE;	
END_IF

CASE nCase OF
	0:
		IF bExecute THEN
			bBusy		:= TRUE;
			nCase 		:= 10;
			nErrorID 	:= 0;
			nCurArrLoc 	:= 1;
			fbCoE_Read(bExecute:=FALSE);
		END_IF
		
		
	10: //Read CoE Address Data
		fbCoE_Read(
			nIndex 		:= stCoEDataArray.stCoEData[nCurArrLoc].nIndex,
			nSubIndex 	:= stCoEDataArray.stCoEData[nCurArrLoc].nSubIndex,
			pDstBuf 	:= ADR(stCoEDataArray.stCoEData[nCurArrLoc].dwData),
			cbBufLen 	:= stCoEDataArray.stCoEData[nCurArrLoc].nDataLen,
			bExecute 	:= TRUE );
			
		IF fbCoE_Read.bError THEN
			nCase	:= 9999;
		ELSIF NOT fbCoE_Read.bBusy THEN
			nCase := 20;
		END_IF
	
		
	20: //Check for End of Array
		IF nCurArrLoc >= nSizeOfArr THEN
			nCase := 10000;
			bDone := TRUE;
		ELSE
			nCurArrLoc := nCurArrLoc + 1;
			nCase := 10;
			fbCoE_Read(bExecute:=FALSE);
		END_IF
		
			
	9999: //Error
		bError 	:= TRUE;
		nErrorID := fbCoE_Read.nErrID;
		fbCoE_Read(bExecute:=FALSE);
		nCase	:= 10000;
		
		
	10000: //Wait for Next 'Execute' Rising Edge
		bBusy := FALSE;
		IF NOT bExecute THEN
			nCase := 0;
		END_IF
		
END_CASE

END_FUNCTION_BLOCK

// ---- POUs/Function Blocks/FB_CoE_WriteParamArray.TcPOU
FUNCTION_BLOCK FB_CoE_WriteParamArray
VAR_INPUT
	bExecute: BOOL;
	sNetId: T_AmsNetID;
	nSlaveAddr: UINT;
	tTimeout: TIME;
	nSizeOfArr: USINT;
END_VAR
VAR_OUTPUT
	bBusy: BOOL;
	bDone: BOOL;
	/// Current ST_CoEDataArray Array Location being Write
	nCurArrLoc: INT;
	bError: BOOL;
	/// http://infosys.beckhoff.com/content/1033/tcadscommon/html/ads_returncodes.htm
	nErrorID: UDINT;
END_VAR
VAR
	fbCoE_Write: FB_EcCoESdoWrite;
	nCase: INT;
	nIndex: INT;
END_VAR
VAR_IN_OUT
	stCoEDataArray: ST_CoEDataArray;
END_VAR

(*++++++++++++++ CoE communication ++++++++++++++++++++++*)
fbCoE_Write.sNetId		:= sNetId;
fbCoE_Write.nSlaveAddr 	:= nSlaveAddr;
fbCoE_Write.tTimeout		:= tTimeout;

//Automatically Resets FB if bExecute is False
IF NOT bExecute THEN
	nCase 		:= 0;
	bError 		:= FALSE;
	bBusy 		:= FALSE;
	bDone 		:= FALSE;	
END_IF

CASE nCase OF
	0:
		IF bExecute THEN
			bBusy		:= TRUE;
			nCase 		:= 10;
			nErrorID 	:= 0;
			nCurArrLoc 	:= 1;
			fbCoE_Write(bExecute:=FALSE);
		END_IF
		
		
	10: //Write CoE Address Data
		fbCoE_Write(
			nIndex 		:= stCoEDataArray.stCoEData[nCurArrLoc].nIndex,
			nSubIndex 	:= stCoEDataArray.stCoEData[nCurArrLoc].nSubIndex,
			pSrcBuf 	:= ADR(stCoEDataArray.stCoEData[nCurArrLoc].dwData),
			cbBufLen 	:= stCoEDataArray.stCoEData[nCurArrLoc].nDataLen,
			bExecute 	:= TRUE );
			
		IF fbCoE_Write.bError THEN
			nCase	:= 9999;
		ELSIF NOT fbCoE_Write.bBusy THEN
			nCase := 20;
		END_IF
	
		
	20: //Check for End of Array
		IF nCurArrLoc >= nSizeOfArr THEN
			nCase := 10000;
			bDone := TRUE;
		ELSE
			nCurArrLoc := nCurArrLoc + 1;
			nCase := 10;
			fbCoE_Write(bExecute:=FALSE);
		END_IF
		
			
	9999: //Error
		bError 	:= TRUE;
		nErrorID := fbCoE_Write.nErrID;
		fbCoE_Write(bExecute:=FALSE);
		nCase	:= 10000;
		
		
	10000: //Wait for Next 'Execute' Rising Edge
		bBusy := FALSE;
		IF NOT bExecute THEN
			nCase := 0;
		END_IF
		
END_CASE

END_FUNCTION_BLOCK

// ---- POUs/Function Blocks/FB_CoE_SaveParam.TcPOU
FUNCTION_BLOCK FB_CoE_SaveParam
VAR_INPUT
	bExecute: BOOL;
	sNetId: T_AmsNetID;
	nSlaveAddr: UINT;
	tTimeout: TIME;
	nSizeOfArr: USINT;
END_VAR
VAR_OUTPUT
	bBusy: BOOL;
	bDone: BOOL;
	
	bError: BOOL;
	/// http://infosys.beckhoff.com/content/1033/tcadscommon/html/ads_returncodes.htm
	nErrorID: UDINT;
	/// http://infosys.beckhoff.com/content/1033/tcadscommon/html/ads_returncodes.htm
END_VAR
VAR
	fbCoE_Write: FB_EcCoESdoWrite;
	fbCoE_Read: FB_EcCoESdoRead;
	
	nCase:	INT;
	nIndex:	INT;
	nSubIndex:	INT;
	nData: INT;
END_VAR

//Issues a SaveAll Command to the Drive to store parameters in case of powerloss

(*++++++++++++++ CoE communication ++++++++++++++++++++++*)
fbCoE_Read.sNetId		:= sNetId;
fbCoE_Read.nSlaveAddr 	:= nSlaveAddr;
fbCoE_Read.tTimeout		:= tTimeout;

fbCoE_Write.sNetId		:= sNetId;
fbCoE_Write.nSlaveAddr 	:= nSlaveAddr;
fbCoE_Write.tTimeout	:= tTimeout;

//Automatically Resets FB if bExecute is False
IF NOT bExecute THEN
	nCase 		:= 0;
	bError 		:= FALSE;
	bBusy 		:= FALSE;
	bDone 		:= FALSE;	
END_IF

CASE nCase OF
	0:
		IF bExecute THEN
			bBusy		:= TRUE;
			nCase 		:= 10;
			nErrorID 	:= 0;
			fbCoE_Write(bExecute:=FALSE);
		END_IF
		
		
	10: //Write CoE Address Data
		fbCoE_Write(
			sNetId:= , 
			nSlaveAddr:= GVL_IO.stAmsAddr_Kid_1.port, 
			nSubIndex:= 16#01, 
			nIndex:= 	16#1010, 
			pSrcBuf:= 	ADR(nData), 
			cbBufLen:= 	SIZEOF(nData), 
			bExecute:= TRUE, 
			tTimeout:= , 
			bBusy=> , 
			bError=> , 
			nErrId=> );

		IF fbCoE_Write.bError THEN
			nCase	:= 9998;
		ELSIF NOT fbCoE_Write.bBusy THEN
			fbCoe_Write(bExecute:=FALSE);
			nCase := 20;
		END_IF
	
	20:	//Read CoE Address Data, place in internal variable
		fbCoE_Read(
			sNetId:= , 
			nSlaveAddr:= GVL_IO.stAmsAddr_Kid_1.port, 
			nSubIndex:= 16#01, 
			nIndex:= 	16#1010, 
			pDstBuf:=	ADR(nData) , 
			cbBufLen:= 	SIZEOF(nData), 
			bExecute:= TRUE, 
			tTimeout:= , 
			bBusy=> , 
			bError=> , 
			nErrId=> );
	
		IF fbCoE_Read.bError THEN
			nCase	:= 9999;
		ELSIF NOT fbCoE_Read.bBusy THEN
			fbCoe_Read(bExecute:=FALSE);
			nCase := 30;
		END_IF	
		
	30:	//Compare that Write & Read data are same, if not then go to Case 10, else go to case 40
		IF fbCoE_Write.pSrcBuf = fbCoE_Read.pDstBuf THEN
			nCase := 40;
		ELSE
			nCase := 10;
		END_IF
	
	40:	//issue a reset command to drive
		//To Do: add a reset drive command
		
	
	
	9998: //Error
		bError 	:= TRUE;
		nErrorID := fbCoE_Write.nErrID;
		fbCoE_Write(bExecute:=FALSE);
		nCase	:= 10000;
	
	9999: //Error
		bError 	:= TRUE;
		nErrorID := fbCoE_Read.nErrID;
		fbCoE_Read(bExecute:=FALSE);
		nCase	:= 10000;
		
	10000:
		
	
END_CASE

END_FUNCTION_BLOCK

// ---- POUs/Function Blocks/FB_stCoEData_Comparison.TcPOU
FUNCTION_BLOCK FB_stCoEData_Comparison
VAR_INPUT
	nNumOfPara	:	INT;
	bExecute: BOOL;
END_VAR
VAR_OUTPUT
	bError	 : BOOL;
	nErrorID : UINT;
	bDone 	 : BOOL;
	
END_VAR
VAR
	nCase : UINT;
	index : UINT;
END_VAR

		//change this to a for-loop to step through each read & write array to verify
		//error codes should kick if it gets stuck
		//if not the same then run INIT again???
		
		//should this be in a Function Block???
	CASE nCase OF
		0:	
			IF bExecute THEN
				bError := FALSE;
				index := 1;
				nCase := 10;
			END_IF
		10:	
			
			WHILE ((index	<= nNumOfPara) AND NOT bError) DO
				
				IF stCoEDataArray_Write.stCoEData[index].dwData <> stCoEDataArray_Read.stCoEData[index].dwData THEN	
					bError := TRUE;
					nErrorID := index;
					nCase :=	9999;
				ELSE
					nCase :=	10000;
				END_IF
				
					index := index + 1;
			END_WHILE
			
		9999:
				
				nCase := 0;
						
		10000:
			bDone := TRUE;
			IF NOT bExecute THEN
				bDone := FALSE;
				nCase := 0;
			END_IF
	END_CASE

END_FUNCTION_BLOCK

// ---- POUs/Function Blocks/FB_WriteLimits.TcPOU
FUNCTION_BLOCK FB_WriteLimits
VAR_INPUT
	bExecute	: BOOL;
	dnUpLimit	: DINT;
	dnDownLimit	: DINT;
END_VAR
VAR_OUTPUT
	
	bDone 		: BOOL;	//both limits were written and verified
	bError		: BOOL; //Error writing or limits not verified
	udnErrorID	: UDINT;	//Error code, to be added to later (writing or reading)
	bBusy		: BOOL;	//in the process of running the Function Blocks

	
END_VAR
VAR
	fbMC_WriteUPParameter: MC_WriteParameter;
	fbMc_WriteDownParameter: MC_WriteParameter;
	WriteLimits: INT;
	fbMC_ReadUPParameter: MC_ReadParameter;
	fbMC_ReadDownParameter: MC_ReadParameter;
END_VAR
VAR_IN_OUT
	Axis		: Axis_Ref;
	
END_VAR

	
CASE WriteLimits OF
	
	0 :	//wait for the bExecute
		IF bExecute THEN
			bError		:= FALSE;
			udnErrorID	:= 0;
			bBusy		:= TRUE;
			WriteLimits := 2;
		END_IF

	2 :	//setting Function Block to False
		fbMC_WriteUPParameter(Axis:= Axis ,Execute:= FALSE);
		WriteLimits := WriteLimits +1;	
		
	3 :	//write to the up limit	
		
		fbMC_WriteUPParameter(		//Execute the Write Parameter for NC
			Axis			:= Axis ,
			Execute			:= TRUE, 
			ParameterNumber	:= AxisMaxSoftPosLimit, 
			Value			:= DINT_TO_LREAL(dnUpLimit), 
			Done			=> , 
			Busy			=> , 
			Error			=> , 
			ErrorID			=> udnErrorID);
		
		IF fbMC_WriteUPParameter.Error THEN
			
			WriteLimits := 9999;
			//Add error handling 
		ELSE
			IF fbMC_WriteUPParameter.Done THEN
				fbMC_WriteUPParameter(Axis:= Axis ,Execute:= FALSE);
				WriteLimits := WriteLimits +1;
			END_IF
		END_IF	
		
	4:	//Setting FB to False
		fbMC_ReadUPParameter(Axis:= Axis ,Enable:= FALSE);
		WriteLimits := WriteLimits +1;	
	
	5:	//Reading last value of UpLimit written in Case 4
		fbMC_ReadUPParameter(
			Axis:= Axis, 
			Enable:= TRUE, 
			ParameterNumber:= AxisMaxSoftPosLimit, 
			ReadMode:= ReadMode_Once, 
			Valid=> , 
			Busy=> , 
			Error=> , 
			ErrorID=> , 
			Value=> );

		IF fbMC_ReadUPParameter.Error THEN
			WriteLimits := 9999;
			//Add error handling 
		ELSE
			IF NOT fbMC_ReadUPParameter.Busy THEN
				fbMC_ReadUPParameter(Axis:= Axis ,Enable:= FALSE);
				WriteLimits := WriteLimits +1;
			END_IF
		END_IF		
			
	6:	//Comparison of Written Value to Read Value
	
		IF fbMC_ReadUPParameter.Value = DINT_TO_LREAL(dnUpLimit) THEN
			WriteLimits := WriteLimits +1;
		ELSE
			WriteLimits := 9999;
		END_IF
		
	7:	//setting Function Block to False
		fbMC_WriteDownParameter(Axis:= Axis ,Execute:= FALSE);
		WriteLimits := WriteLimits +1;	
		
	8 :	//write to the down limit	
		
		fbMC_WriteDownParameter(		//Execute the Write Parameter for NC
			Axis			:= Axis ,
			Execute			:= TRUE, 
			ParameterNumber	:= AxisMinSoftPosLimit, 
			Value			:= DINT_TO_LREAL(dnDownLimit), 
			Done			=> , 
			Busy			=> , 
			Error			=> , 
			ErrorID			=> udnErrorID);
		
		IF fbMC_WriteDownParameter.Error THEN
			
			WriteLimits := 9999;
			//Add error handling 
		ELSE
			IF fbMC_WriteDownParameter.Done THEN
				fbMC_WriteDownParameter(Axis:= Axis ,Execute:= FALSE);
				WriteLimits := WriteLimits +1;
			END_IF
		END_IF	
		
	9:	//Setting FB to False
		fbMC_ReadDownParameter(Axis:= Axis ,Enable:= FALSE);
		WriteLimits := WriteLimits +1;	
	
	10:	//Reading last value of UpLimit written in Case 4
		fbMC_ReadDownParameter(
			Axis:= Axis, 
			Enable:= TRUE, 
			ParameterNumber:= AxisMinSoftPosLimit, 
			ReadMode:= ReadMode_Once, 
			Valid=> , 
			Busy=> , 
			Error=> , 
			ErrorID=> , 
			Value=> );

		IF fbMC_ReadDownParameter.Error THEN
			WriteLimits := 9999;
			//Add error handling 
		ELSE
			IF NOT fbMC_ReadDownParameter.Busy THEN
				fbMC_ReadDownParameter(Axis:= Axis ,Enable:= FALSE);
				WriteLimits := WriteLimits +1;
			END_IF
		END_IF		
			
	11:	//Comparison of Written Value to Read Value
	
		IF fbMC_ReadDownParameter.Value = DINT_TO_LREAL(dnDownLimit) THEN
			fbMC_WriteUPParameter(Axis := Axis, Execute := FALSE);
			WriteLimits := WriteLimits +1;
		ELSE
			WriteLimits := 9999;
		END_IF
	
	12: //Verify that Soft Limit Switch is enabled
	
	fbMC_WriteUPParameter(		//Execute the Write Parameter for NC
			Axis			:= Axis ,
			Execute			:= TRUE, 
			ParameterNumber	:= AxisEnMaxSoftPosLimit, 
			Value			:= BOOL_TO_LREAL(TRUE), 
			Done			=> , 
			Busy			=> , 
			Error			=> , 
			ErrorID			=> udnErrorID);
		
		IF fbMC_WriteUPParameter.Error THEN
			
			WriteLimits := 9999;
			//Add error handling 
		ELSE
			IF fbMC_WriteUPParameter.Done THEN
				fbMC_WriteUPParameter(Axis:= Axis ,Execute:= FALSE);
				WriteLimits := WriteLimits +1;
			END_IF
		END_IF	
		
	13:	//Setting FB to False
		fbMC_ReadUPParameter(Axis:= Axis ,Enable:= FALSE);
		WriteLimits := WriteLimits +1;	
	
	14:	//Reading last value of UpLimit written in Case 4
		fbMC_ReadUPParameter(
			Axis:= Axis, 
			Enable:= TRUE, 
			ParameterNumber:= AxisEnMaxSoftPosLimit, 
			ReadMode:= ReadMode_Once, 
			Valid=> , 
			Busy=> , 
			Error=> , 
			ErrorID=> , 
			Value=> );

		IF fbMC_ReadUPParameter.Error THEN
			WriteLimits := 9999;
			//Add error handling 
		ELSE
			IF NOT fbMC_ReadUPParameter.Busy THEN
				fbMC_ReadUPParameter(Axis:= Axis ,Enable:= FALSE);
				WriteLimits := WriteLimits +1;
			END_IF
		END_IF		
			
	15:	//Comparison of Written Value to Read Value
	
		IF fbMC_ReadUPParameter.Value = BOOL_TO_LREAL(TRUE) THEN
			WriteLimits := WriteLimits +1;
		ELSE
			WriteLimits := 9999;
		END_IF
		
	16:	//setting Function Block to False
		fbMC_WriteDownParameter(Axis:= Axis ,Execute:= FALSE);
		WriteLimits := WriteLimits +1;
		
	17:	//write to the down limit	
		
		fbMC_WriteDownParameter(		//Execute the Write Parameter for NC
			Axis			:= Axis ,
			Execute			:= TRUE, 
			ParameterNumber	:= AxisEnMinSoftPosLimit, 
			Value			:= BOOL_TO_LREAL(TRUE), 
			Done			=> , 
			Busy			=> , 
			Error			=> , 
			ErrorID			=> udnErrorID);
		
		IF fbMC_WriteDownParameter.Error THEN
			
			WriteLimits := 9999;
			//Add error handling 
		ELSE
			IF fbMC_WriteDownParameter.Done THEN
				fbMC_WriteDownParameter(Axis:= Axis ,Execute:= FALSE);
				WriteLimits := WriteLimits +1;
			END_IF
		END_IF	
		
	18:	//Setting FB to False
		fbMC_ReadDownParameter(Axis:= Axis ,Enable:= FALSE);
		WriteLimits := WriteLimits +1;
	
	19:	//Reading last value of UpLimit written in Case 4
		fbMC_ReadDownParameter(
			Axis:= Axis, 
			Enable:= TRUE, 
			ParameterNumber:= AxisEnMinSoftPosLimit, 
			ReadMode:= ReadMode_Once, 
			Valid=> , 
			Busy=> , 
			Error=> , 
			ErrorID=> , 
			Value=> );

		IF fbMC_ReadDownParameter.Error THEN
			WriteLimits := 9999;
			//Add error handling 
		ELSE
			IF NOT fbMC_ReadDownParameter.Busy THEN
				fbMC_ReadDownParameter(Axis:= Axis ,Enable:= FALSE);
				WriteLimits := WriteLimits +1;
			END_IF
		END_IF		
			
	20:	//Comparison of Written Value to Read Value
	
		IF fbMC_ReadDownParameter.Value = BOOL_TO_LREAL(TRUE) THEN
			WriteLimits := 10000;
		ELSE
			WriteLimits := 9999;
		END_IF

	
	9999:	//Error Handling
		bError  := TRUE;
		bBusy	:= FALSE;
				
		IF NOT bExecute THEN
			WriteLimits := 0;
		END_IF	
	
	10000:	//Done writing and verifying limits
		bBusy	:= FALSE;
		bDone	:= TRUE;
		
		IF NOT bExecute THEN
			WriteLimits := 0;
			bDone		:= false;
		END_IF	
		
END_CASE

END_FUNCTION_BLOCK

// ---- POUs/Function Blocks/FB_IgnoreLimits.TcPOU
FUNCTION_BLOCK FB_IgnoreLimits
VAR_INPUT
	bExecute	: BOOL;
	bLimit_Use	: BOOL;
END_VAR
VAR_OUTPUT
	
	bDone 		: BOOL;	//both limits were written and verified
	bError		: BOOL; //Error writing or limits not verified
	udnErrorID	: UDINT;	//Error code, to be added to later (writing or reading)
	bBusy		: BOOL;	//in the process of running the Function Blocks

	
END_VAR
VAR
	fbMC_WriteUPParameter	: MC_WriteParameter;
	fbMc_WriteDownParameter	: MC_WriteParameter;
	WriteLimits				: INT;
	fbMC_ReadUPParameter	: MC_ReadParameter;
	fbMC_ReadDownParameter	: MC_ReadParameter;
END_VAR
VAR_IN_OUT
	Axis		: Axis_Ref;
	
END_VAR

	
CASE WriteLimits OF
	
	0 :	//wait for the bExecute
		IF bExecute THEN
			bError		:= FALSE;
			udnErrorID	:= 0;
			bBusy		:= TRUE;
			WriteLimits := 2;
			
		END_IF

	2 :	//setting Function Block to False
		fbMC_WriteUPParameter(Axis:= Axis ,Execute:= FALSE);
		WriteLimits := 3;	
		
	3 :	//set the Up Limit Switch Enable to "OFF"	
		
		fbMC_WriteUPParameter(		//Execute the Write Parameter for NC
			Axis			:= Axis ,
			Execute			:= TRUE, 
			ParameterNumber	:= AxisEnMaxSoftPosLimit, 
			Value			:= BOOL_TO_LREAL(bLimit_Use), 
			Done			=> , 
			Busy			=> , 
			Error			=> , 
			ErrorID			=> udnErrorID);
		
		IF fbMC_WriteUPParameter.Error THEN
			
			WriteLimits := 9999;
			//Add error handling 
		ELSE
			IF fbMC_WriteUPParameter.Done THEN
				fbMC_WriteUPParameter(Axis:= Axis ,Execute:= FALSE);
				WriteLimits := 4;
			END_IF
		END_IF	
		
	4:	//Setting FB to False
		fbMC_ReadUPParameter(Axis:= Axis ,Enable:= FALSE);
		WriteLimits := 5;	
	
	5:	//Reading last value of UpLimit written in Case 4
		fbMC_ReadUPParameter(
			Axis:= Axis, 
			Enable:= TRUE, 
			ParameterNumber:= AxisEnMaxSoftPosLimit, 
			ReadMode:= ReadMode_Once, 
			Valid=> , 
			Busy=> , 
			Error=> , 
			ErrorID=> , 
			Value=> );

		IF fbMC_ReadUPParameter.Error THEN
			WriteLimits := 9999;
			//Add error handling 
		ELSE
			IF NOT fbMC_ReadUPParameter.Busy THEN
				fbMC_ReadUPParameter(Axis:= Axis ,Enable:= FALSE);
				WriteLimits := 6;
			END_IF
		END_IF		
			
	6:	//Comparison of Written Value to Read Value
	
		IF fbMC_ReadUPParameter.Value = BOOL_TO_LREAL(bLimit_Use) THEN
			WriteLimits := 7;
		ELSE
			WriteLimits := 9999;
		END_IF
		
	7:	//setting Function Block to False
		fbMC_WriteDownParameter(Axis:= Axis ,Execute:= FALSE);
		WriteLimits := 8;	
		
	8 :	//write to the down limit	
		
		fbMC_WriteDownParameter(		//Execute the Write Parameter for NC
			Axis			:= Axis ,
			Execute			:= TRUE, 
			ParameterNumber	:= AxisEnMinSoftPosLimit, 
			Value			:= BOOL_TO_LREAL(bLimit_Use), 
			Done			=> , 
			Busy			=> , 
			Error			=> , 
			ErrorID			=> udnErrorID);
		
		IF fbMC_WriteDownParameter.Error THEN
			
			WriteLimits := 9999;
			//Add error handling 
		ELSE
			IF fbMC_WriteDownParameter.Done THEN
				fbMC_WriteDownParameter(Axis:= Axis ,Execute:= FALSE);
				WriteLimits := 9;
			END_IF
		END_IF	
		
	9:	//Setting FB to False
		fbMC_ReadDownParameter(Axis:= Axis ,Enable:= FALSE);
		WriteLimits := 10;	
	
	10:	//Reading last value of UpLimit written in Case 4
		fbMC_ReadDownParameter(
			Axis:= Axis, 
			Enable:= TRUE, 
			ParameterNumber:= AxisEnMinSoftPosLimit, 
			ReadMode:= ReadMode_Once, 
			Valid=> , 
			Busy=> , 
			Error=> , 
			ErrorID=> , 
			Value=> );

		IF fbMC_ReadDownParameter.Error THEN
			WriteLimits := 9999;
			//Add error handling 
		ELSE
			IF NOT fbMC_ReadDownParameter.Busy THEN
				fbMC_ReadDownParameter(Axis:= Axis ,Enable:= FALSE);
				WriteLimits := 11;
			END_IF
		END_IF		
			
	11:	//Comparison of Written Value to Read Value
	
		IF fbMC_ReadDownParameter.Value = BOOL_TO_LREAL(bLimit_Use) THEN
			WriteLimits := 10000;
		ELSE
			WriteLimits := 9999;
		END_IF
		
	9999:	//Error Handling
		bError  := TRUE;
		bBusy	:= FALSE;
				
		IF NOT bExecute THEN
			WriteLimits := 0;
		END_IF	
	
	10000:	//Done writing and verifying limits
		bBusy	:= FALSE;
		bDone	:= TRUE;
		
		IF NOT bExecute THEN
			WriteLimits := 0;
			bDone		:= false;
		END_IF	
		
END_CASE

END_FUNCTION_BLOCK

// ---- POUs/Functions/F_Scale_LR.TcPOU
FUNCTION F_Scale_LR : LREAL
VAR_INPUT
	
	lrInputWeight		:	LREAL;	//Weight (g) actual weight
	lrMinWeight			:	LREAL; 	//Weight (g)
	lrMaxWeight			:	LREAL;	//Weight (g)
	lrAtMinWeight		:	LREAL;	//Min Accel/decel value (mm/s2)
	lrAtMaxWeight		:	LREAL;	//Max Accel/Decel value (mm/s2)
	bLimitOutput		:	BOOL;	//Is the function Used?
	
END_VAR
VAR
	lrValue: LREAL;
END_VAR




//NewInputValue is Scaled between the min & max output values
//
IF 	lrMinWeight 		< 0 OR
	lrMaxWeight			<= 0 OR
	lrAtMinWeight	<= 0 OR
	lrAtMaxWeight	<= 0 THEN
	lrValue := 0;
ELSIF lrInputWeight < lrMinWeight THEN
	lrValue	:= lrAtMinWeight;

ELSE
	IF bLimitOutput = TRUE THEN
		lrValue 	:=	(((lrMaxWeight - lrInputWeight) / lrMaxWeight) * (lrAtMinWeight) )  ;
		IF lrValue	< lrAtMaxWeight THEN
			lrValue	:= lrAtMaxWeight;
		END_IF
	ELSE
		lrValue :=	lrAtMinWeight;	
	END_IF
END_IF

F_Scale_LR	:= lrValue;

END_FUNCTION

// ---- POUs/Programs/EtherCAT/FB_CheckIn_EtherCAT.TcPOU
FUNCTION_BLOCK FB_CheckIn_EtherCAT
VAR_INPUT
		QuickPressTimer : INT;
		QuickPressCounter : INT;
		VoltageEnabledCounter : DINT;
		KidID : INT;
		Home_Tripped : BOOL;
			momControl: BOOL; //flag used to indicate if targets are taken from mom or Joystick

END_VAR
VAR_OUTPUT
	JoyStickMode : BOOL;

	MomEstopActivated : BOOL;
	Rmt_DeadManPressed : BOOL;
	Rmt_CollisionDetect : BOOL;
	Unknown: BOOL;
	heartBeat : BOOL;
	ComError_Reset : BOOL; //Used both to indicate a Comm_Error(FromKid) and reset a Comm_Error(ToKid)
	Mom_System_Estop: BOOL;
	ResetSaftey : BOOL;
	SafteyTripped : BOOL;
	Hard_Limit_Tripped : BOOL;
	SetSoftUp : BOOL;
	SetSoftDown : BOOL;
END_VAR
VAR
	checkingInt : UDINT;
	checkint1 : DINT;
	//Heartbeat for timeout and COMS over EtherCAT
	MomComTimer : TON; //Starts timer if a cycle heartbeat is missed. 100MS = COMLOSS
	MomCom_ET : TIME; //Elapsed Time since last update
	HomeOperation_Active : BOOL;
END_VAR

IF GVL_Hardware_IO.bLocal_Deadman_State THEN 
	QuickPressTimer := QuickPressTimer + 1;
	IF QuickPressTimer > 50 THEN QUickpressCounter := 0; quickpressTimer :=50; END_IF
	ELSIF QuickPressTimer < 50 AND quickpressTimer > 0 THEN
		QuickPressCounter := QuickpressCounter + 1;
		IF QuickPressCounter > 10 THEN 
			GVL_Safe_IO.bSafetySystem_Reset := TRUE; 
			gvl_hmi.momcontrol_bypass := QuickPressCounter < 15 ;
			 
		END_IF
		quickpressTimer := 0;
		ELSE
			
		quickpresstimer:=0;
END_IF

IF GVL_HMI.MomControl_Bypass THEN 
	IF MomControl THEN GVL_Safe_IO.bSafetySystem_Reset := TRUE; END_IF
	 MomEstopActivated := FALSE; 
	 momControl := FALSE;
	 KidAxis.UpdateWord_toMom := (KidID * 2048) + (BOOL_TO_UINT(momControl)* 128);
	RETURN; 
END_IF

checkingInt := KidAxis.UpdateWord_FromMom;
 	
	IF CheckIngInt/134217728 > 0 THEN KidID := UDINT_TO_INT(CheckingInt / 134217728); checkingInt := CheckingInt MOD 134217728; END_IF
	checkingInt := CheckingInt MOD 4096; 
	IF CheckingInt/512 > 0 AND NOT HomeOperation_Active AND NOT (checkingInt MOD 16)/8 >0 THEN
		GVL_Safe_IO.bHard_Up_Bypass_Enable := TRUE;
		GVL_Safe_IO.bHard_Down_Bypass_Enable := TRUE;
	ELSIF CheckingInt/512 = 0 AND HomeOperation_Active AND NOT (checkingInt MOD 16)/8 >0 THEN
		GVL_Safe_IO.bHard_Up_Bypass_Enable := FALSE;
		GVL_Safe_IO.bHard_Down_Bypass_Enable := FALSE;
		GVL_Index.Home_Offset := Kidaxis.actualPos + GVL_Index.Home_Switch_Offset;
		GVL_Index.Home_Offset_UU := GVL_Index.Home_Offset / LREAL_TO_INT(1/ GVL_Motion.lrEncoder_ScalingNum);

		//IF GVL_Index.Home_Offset < GVL_Index.Admin_Min THEN GVL_Index.Admin_Min := GVL_Index.Home_Offset ; END_IF
	END_IF
	//IF KidID = 0 THEN RETURN; END_IF
	KidAxis.byPassSoftDown := CheckingInt/16384 >0; checkingInt := checkingInt MOD 1024;
	KidAxis.byPassSoftUp := CheckingInt/8192 >0; checkingInt := checkingInt MOD 1024;
	KidAxis.byPassHardDown := CheckingInt/4096 >0; checkingInt := checkingInt MOD 1024;
	KidAxis.byPassHardUp := CheckingInt/2048 >0; checkingInt := checkingInt MOD 1024;
	KidAxis.byPassUltimate := CheckingInt/1024 >0; checkingInt := checkingInt MOD 1024;
	HomeOperation_Active := CheckingInt/512 > 0; checkingInt := checkingInt MOD 512;
	Rmt_CollisionDetect :=CheckingInt/256 > 0; checkingInt := CheckingInt MOD 256;
	momControl:= checkingInt / 128 > 0 ;	checkingInt := checkingInt MOD 128;
	Rmt_DeadManPressed:= checkingInt / 64 > 0;	checkingInt := checkingInt MOD 64;
	ResetSaftey := checkingInt / 32 > 0;	checkingInt := checkingInt MOD 32;
	ComError_Reset:= checkingInt / 16 > 0;	checkingInt := checkingInt MOD 16;
	MomEstopActivated:= checkingInt / 8 > 0;	checkingInt := checkingInt MOD 8;
	JoyStickMode:= checkingInt / 4 > 0;	checkingInt := checkingInt MOD 4;
	KidAxis.LeaveEnabled:= checkingInt / 2 > 0;   checkingInt := checkingInt MOD 2;
	HeartBeat :=CheckingInt>0;

IF ComError_Reset OR ResetSaftey THEN
	GVL_PLC.bGLOBAL_ERROR_STRING := replace(GVL_PLC.bGlobal_Error_String, '', len('Comm Lost on EtherCat Network'), FIND(GVL_PLC.bGLOBAL_ERROR_STRING, 'Comm Lost on EtherCat Network'));
	MomComTimer.IN := FALSE;
GVL_PLC.bComTimeOutError := FALSE;
	MomComTimer.PT := T#2S;
	
END_IF

		
IF  NOT GVL_PLC.bComTimeOutError OR ComError_Reset THEN
MomComTimer(IN:=HeartBeat, PT:=T#150MS , Q=>GVL_PLC.bComTimeOutError, ET=> MomCom_ET ); //Starts timer if a cycle heartbeat is missed. 100MS = COMLOSS
ELSE
	
	IF FIND(GVL_PLC.bGLOBAL_ERROR_STRING, 'Comm Lost on EtherCat Network')=0 THEN
		GVL_PLC.bGLOBAL_ERROR_STRING := CONCAT(GVL_PLC.bGlobal_Error_String, 'Comm Lost on EtherCat Network');
	END_IF
	
END_IF

IF ResetSaftey THEN
	GVL_Safe_IO.bSafetySystem_Reset := TRUE;
	MomEstopActivated := FALSE;
	VoltageEnabledCounter := 100;
END_IF
		IF NOT KidAxis.Status.STATve AND NOT ResetSaftey THEN 
			IF VoltageENabledCounter > -100 THEN VoltageENabledCounter := VoltageEnabledCounter - 1; END_IF
		ELSIF KidAxis.Status.STATve THEN
			IF VoltageENabledCounter < 100 THEN VoltageENabledCounter := VoltageEnabledCounter + 1; END_IF
		END_IF
		
SafteyTripped := NOT bPlcEstopSignal OR  Kidaxis.Status.statf OR GVL_PLC.bComTimeOutError OR NOT GVL_Safe_IO.bContactor OR VoltageEnabledCounter < -15; 
Hard_Limit_Tripped := NOT bLimit_Hard_Up OR NOT bLimit_Hard_Down;
KidAxis.UpdateWord_toMom := INT_TO_UDINT(KidID) * 134217728 +

BOOL_TO_UDINT(KIDAXIS.modeTargetPos < gvl_iNDEX.Admin_MIN) * 16384 +
BOOL_TO_UDINT(KIDAXIS.modeTargetPos > gvl_iNDEX.Admin_Max) * 8192 +
BOOL_TO_UDINT(gvl_sAFE_io.bLimit_Hard_Down) * 4096 +
BOOL_TO_UDINT(gvl_sAFE_io.bLimit_Hard_uP) * 2048 +
BOOL_TO_UDINT(gvl_sAFE_io.bLimiT_uLTIMATE) * 1024 +
										BOOL_TO_UDINT(NOT GVL_Safe_IO.bES_Local_Status) * 512 +
										BOOL_TO_UDINT(momControl) * 128 +
										BOOL_TO_UDINT(GVL_Safe_IO.bSlack_Line) * 64 +
										BOOL_TO_UDINT(Kidaxis.Status.voltageEnabled) * 32 +
										BOOL_TO_UDINT(GVL_PLC.bComTimeOutError) * 16 +
										BOOL_TO_UDINT(SafteyTripped) * 8 +
										BOOL_TO_UDINT(Hard_Limit_Tripped) * 4 +
										BOOL_TO_UDINT(kidAxis.LeaveEnabled) * 2 +
										BOOL_TO_UDINT(NOT HeartBeat);
						
			momControl := momControl AND NOT GVL_PLC.bComTimeOutError ;					
IF (momControl OR ResetSaftey) AND NOT ((MomEstopActivated AND momControl) OR (GVL_PLC.bComTimeOutError AND momControl)) THEN 
	
		GVL_Modes.nMotion_Command := 10;

ELSE
	GVL_Modes.nMotion_Command := 2;
END_IF

ResetSaftey := ResetSaftey AND SafteyTripped;

checkint1:= checkint1 + 1;

END_FUNCTION_BLOCK

// ---- POUs/Programs/EtherCAT/FB_EtherCATReader.TcPOU
FUNCTION_BLOCK FB_EtherCATReader
VAR_INPUT
		ID : USINT;
END_VAR
VAR_OUTPUT
	WrittenAll : BOOL := FALSE;
END_VAR

VAR
	SymInfo  : PLC_ReadSymInfo;
	VarSymInfo  :  PLC_ReadSymInfoByName;
	Exec : BOOL;
	
	DataInt : DINT;
	//RecievedData : ARRAY [1..256] OF INT; //used to count reads of each parameter
	i : INT;
	ParametersWritten : USINT;
	RefreshParameters : BOOL := FALSE;
	
	ParameterID_FromMom AT %I* : USINT;
	ParameterWord_FromMom AT %I* : DINT; //ParameterWord cycles through many arrays to send less time critical data
	ParameterID_ToMom AT %Q* : USINT;
END_VAR

//ParameterWord_FromMom consists of 32 bytes. The first(greatest) 8 bytes ID the Variable to write and the last 24 include the data. 
// ParameterID		Parameter To Write					Format
// 1				GVL_Motion.lrEncoder_ScalingNum		1/DATAINT := ScalingNum
// 2				GVL_Index.Admin_Max					:= 512 * DataInt (largest bit is sign)	
// 3				GVL_Index.Admin_Min					:= 	512 * DataInt (largest bit is sign)	
// 4				GVL_Index.Direction_Flipped			>0 		
// 5				GVL_Motion.lrDistance_1_Motor_Rev	:= ?????????????????????????
// 6				GVL_Speeds.QuickStop_Accel		
// 7 				GVL_Speeds.lrDecel_For_EStop		:=?
SymInfo(Port:=851, Start:=Exec);
VarSymInfo(Port:=851, SymName:= 'P30_MAIN.execute', Start:=Exec);

DataInt := Parameterword_FromMom ;
ID := ParameterID_FromMom ;

CASE ID OF
//1: 	GVL_Motion.lrEncoder_ScalingNum := 1/DINT_TO_LREAL(DataInt);
2: 	GVL_Index.Home_Switch_Offset := DataInt ;
3: 	GVL_Index.Admin_Min :=  DataInt ;
4:  GVL_Index.Direction_Flipped := DataInt > 0;
5: 	GVL_Motion.lrDistance_1_Motor_Rev := DataInt;
//6:	GVL_Speeds.QuickStop_Accel := DataInt;
//7:	GVL_Speeds.lrDecel_For_EStop := DataInt;
	
ELSE
	ID := 0;
END_CASE

ParameterID_ToMom := ParameterID_FromMom;

//RecievedData[ID] := RecievedData[ID] + 1;

ParametersWritten := 0;
FOR i := 1 TO 256 DO
//	IF RefreshParameters THEN RecievedData[i] := 0;  END_IF	
	//IF RecievedData[i] > 0 THEN ParametersWritten := ParametersWritten + 1; END_IF
END_FOR

IF RefreshParameters THEN RefreshParameters := FALSE; END_IF

END_FUNCTION_BLOCK

// ---- POUs/Programs/EtherCAT/FB_INIT_EtherCAT.TcPOU
FUNCTION_BLOCK FB_INIT_EtherCAT
VAR_INPUT
END_VAR
VAR_OUTPUT
	Busy: BOOL;
	Disabled: BOOL;
	
		Error: BOOL;
		Moving: BOOL;
		STATf: BOOL;
	//	notMoving: BOOL;
		switchOnDisabled: BOOL;
		voltageEnabled: BOOL;
		STAToe: BOOL;
			STATve: BOOL;
	STATso: BOOL;
		Ready : BOOL;
END_VAR
VAR
   	checkingInt: BITARR16;
	STATha: BOOL;
	STATila: BOOL;
	STATtr: BOOL;
	STATrm: BOOL;
	STATms: BOOL;
	STATw: BOOL;
	STATsod: BOOL;
	STATqs: BOOL;


	
	STATrtso: BOOL;
   //     bExecute                : BOOL; (* rising edge starts writing to the CoE Object *)
    //    bError          : BOOL;
    //    nErrId          : UDINT;
	//	dwData 		: WORD := 16#002;
		nCounter : UINT;
	//	DecelCheckVal : WORD := 16#05;
	//	AccelCheckVal : WORD := 16#05;
		
//		fb_CoEWriteDecel: FB_EcCoESdoWrite;
//	fb_CoEWriteAccel: FB_EcCoESdoWrite;
//	fb_CoEReadAccel : FB_EcCOESDORead;
//	fb_CoEReadDecel : FB_EcCOESDORead;
	
END_VAR

	Error:=TRUE;
checkingInt := kidAxis.statusWord ;
 	STATha:=  checkingint / 4096  > 0; checkingInt := checkingInt MOD 4096;
 	STATila:= checkingInt / 2048 > 0;  checkingInt := checkingInt MOD 2048;
	STATtr:= checkingInt / 1024 > 0;	checkingInt := checkingInt MOD 1024;
	STATrm:= checkingInt / 512 > 0;	checkingInt := checkingInt MOD 512;
	STATms:= checkingInt / 256 > 0;	checkingInt := checkingInt MOD 256;
	STATw:= checkingInt / 128 > 0;	checkingInt := checkingInt MOD 128;
	STATsod:= checkingInt / 64 > 0;	checkingInt := checkingInt MOD 64;
	STATqs:= checkingInt / 32 > 0;	checkingInt := checkingInt MOD 32;
	STATve:= checkingInt / 16 > 0;	checkingInt := checkingInt MOD 16;
	STATf:= checkingInt / 8 > 0;	checkingInt := checkingInt MOD 8;
	STAToe:= checkingInt / 4 > 0;	checkingInt := checkingInt MOD 4;
	STATso:= checkingInt / 2 > 0;   checkingInt := checkingInt MOD 2;
	STATrtso:= checkingInt  > 0;
	Disabled := NOT StatOE;
	//Fault := STATf;
	Moving := STATtr AND kidAxis.isBusy;	
	switchOnDisabled:=STATsod;
	VoltageEnabled := STATve;
	Ready := STATVE AND STATso AND NOT Busy;
	Error:=FALSE;
	
checkingInt := kidaxis.ErrorCode;
	

nCounter := nCounter + 1;

IF  kidaxis.statusWord> 600 THEN	
		KidAxis.OpModeCMD :=2;
		GVL_DriveParameters.controlWord := 270;
		//GVL_DriveParameters.controlWord := 128; //Send HALT command to enable switch on
ELSIF KidAxis.OpModeAct <>2 AND KidAxis.OpModeAct <>0 THEN
		KidAxis.OpModeCMD :=2;
ELSIF StatF THEN
		GVL_DriveParameters.controlWord := 128;
ELSIF kidAxis.status.STATrtso AND NOT kidAxis.status.STATso THEN
		GVL_DriveParameters.controlWord:= 7;

//GVL_DriveParameters.controlWord:= 7;
END_IF

END_FUNCTION_BLOCK

// ---- POUs/Programs/EtherCAT/FB_MoveAbsolute_EtherCAT.TcPOU
 FUNCTION_BLOCK FB_MoveAbsolute_EtherCAT //used to move axis to specified position. 
VAR_INPUT
DeadCounter :Dint ;
END_VAR

